KUKA KRL program: MyProgram_326().src

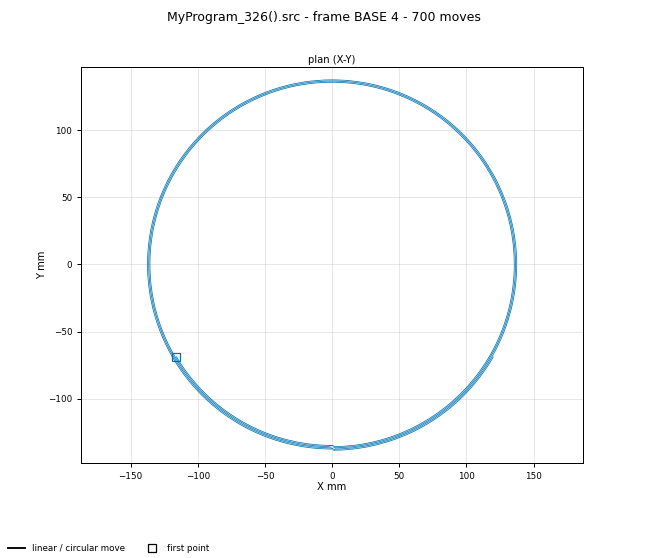
[picture p0: tool path of MyProgram_326().src in frame BASE 4, 700 of 700 moves have a stored position in this frame; points joined in program order, loops and branches not executed]
&ACCESS RVP
&REL 1
&PARAM TEMPLATE = C:\KRC\Roboter\Template\vorgabe
&PARAM EDITMASK = *
DEF MyProgram_326()
; ---- Setting reference (Base) ----
$BASE = BASE_DATA[4]

; --------------------------
; ---- Setting tool (TCP) ----
$TOOL = TOOL_DATA[3]
; --------------------------

$VEL.CP = VEL_APROX_PRINT
Startdeposition()
$VEL.CP = VEL_PRINT
LIN {X -115.9349,Y -68.7238,Z 187,A -143.6936,B 2.3952,C 0.2174,E1 2.2694,E2 236.7794} C_DIS
LIN {X -113.7532,Y -72.2781,Z 187,A -141.7842,B 2.3949,C 0.2211,E1 2.2723,E2 234.8528} C_DIS
LIN {X -111.2945,Y -76.0091,Z 187,A -139.8146,B 2.3945,C 0.2252,E1 2.2754,E2 232.8747} C_DIS
LIN {X -108.8442,Y -79.4786,Z 187,A -137.9392,B 2.3942,C 0.229,E1 2.2785,E2 230.9906} C_DIS
LIN {X -106.312,Y -82.8349,Z 187,A -136.0382,B 2.3938,C 0.2325,E1 2.2817,E2 229.0753} C_DIS
LIN {X -103.5544,Y -86.2576,Z 187,A -134.0833,B 2.3935,C 0.2361,E1 2.2852,E2 227.1095} C_DIS
LIN {X -101.6499,Y -88.4933,Z 187,A -132.7971,B 2.3932,C 0.2385,E1 2.2876,E2 225.8186} C_DIS
LIN {X -98.2627,Y -92.2405,Z 187,A -130.5399,B 2.3928,C 0.2423,E1 2.2919,E2 223.5473} C_DIS
LIN {X -95.1682,Y -95.4297,Z 187,A -128.6658,B 2.3925,C 0.2459,E1 2.2955,E2 221.6755} C_DIS
LIN {X -92.3122,Y -98.195,Z 187,A -126.8323,B 2.3922,C 0.2485,E1 2.2993,E2 219.8233} C_DIS
LIN {X -88.9634,Y -101.2395,Z 187,A -124.8002,B 2.3919,C 0.2515,E1 2.3036,E2 217.7772} C_DIS
LIN {X -85.547,Y -104.1421,Z 187,A -122.818,B 2.3916,C 0.2544,E1 2.3078,E2 215.785} C_DIS
LIN {X -81.9072,Y -107.0279,Z 187,A -120.8161,B 2.3913,C 0.2574,E1 2.3123,E2 213.7795} C_DIS
LIN {X -78.1832,Y -109.778,Z 187,A -118.865,B 2.3909,C 0.2605,E1 2.3167,E2 211.8306} C_DIS
LIN {X -75.0371,Y -111.952,Z 187,A -117.1257,B 2.3907,C 0.2623,E1 2.3207,E2 210.0763} C_DIS
LIN {X -71.5976,Y -114.1827,Z 187,A -115.4752,B 2.3904,C 0.2651,E1 2.3246,E2 208.438} C_DIS
LIN {X -68.7293,Y -115.9316,Z 187,A -113.528,B 2.3904,C 0.2648,E1 2.3294,E2 206.422} C_DIS
LIN {X -65.4366,Y -117.8212,Z 187,A -112.1847,B 2.3901,C 0.2678,E1 2.3326,E2 205.1144} C_DIS
LIN {X -61.68,Y -119.8297,Z 187,A -110.3476,B 2.3899,C 0.2698,E1 2.3372,E2 203.2735} C_DIS
LIN {X -58.7156,Y -121.3102,Z 187,A -108.8853,B 2.3898,C 0.271,E1 2.3409,E2 201.804} C_DIS
LIN {X -55.1373,Y -122.9761,Z 187,A -107.3291,B 2.3895,C 0.2732,E1 2.3448,E2 200.2636} C_DIS
LIN {X -52.5704,Y -124.0969,Z 187,A -105.9692,B 2.3895,C 0.2736,E1 2.3484,E2 198.881} C_DIS
LIN {X -49.184,Y -125.4763,Z 187,A -104.5101,B 2.3893,C 0.2753,E1 2.3521,E2 197.4343} C_DIS
LIN {X -45.9049,Y -126.7124,Z 187,A -103.0422,B 2.3891,C 0.2766,E1 2.356,E2 195.9689} C_DIS
LIN {X -42.7913,Y -127.7975,Z 187,A -101.597,B 2.3891,C 0.2774,E1 2.3598,E2 194.5176} C_DIS
LIN {X -40.0237,Y -128.6924,Z 187,A -100.359,B 2.3889,C 0.2782,E1 2.3631,E2 193.2791} C_DIS
LIN {X -36.5749,Y -129.7136,Z 187,A -98.7075,B 2.3889,C 0.2785,E1 2.3676,E2 191.611} C_DIS
LIN {X -32.9446,Y -130.6827,Z 187,A -97.0537,B 2.3889,C 0.2791,E1 2.3721,E2 189.9491} C_DIS
LIN {X -28.7479,Y -131.6698,Z 187,A -95.2714,B 2.3887,C 0.2801,E1 2.3769,E2 188.173} C_DIS
LIN {X -25.8135,Y -132.2771,Z 187,A -94.096,B 2.3887,C 0.2811,E1 2.3801,E2 187.0102} C_DIS
LIN {X -22.474,Y -132.8846,Z 187,A -92.5645,B 2.3887,C 0.2811,E1 2.3844,E2 185.4665} C_DIS
LIN {X -19.2693,Y -133.3868,Z 187,A -91.2519,B 2.3885,C 0.2817,E1 2.388,E2 184.1621} C_DIS
LIN {X -16.6253,Y -133.7436,Z 187,A -89.7338,B 2.3888,C 0.2798,E1 2.3923,E2 182.5925} C_DIS
LIN {X -11.5747,Y -134.2737,Z 187,A -87.959,B 2.3885,C 0.282,E1 2.3972,E2 180.868} C_DIS
LIN {X -8.5498,Y -134.5003,Z 187,A -86.5532,B 2.3885,C 0.2813,E1 2.4011,E2 179.4461} C_DIS
LIN {X -4.5816,Y -134.6953,Z 187,A -84.6494,B 2.3887,C 0.28,E1 2.4065,E2 177.513} C_DIS
LIN {X 0.9674,Y -134.7656,Z 187,A -83.2917,B 2.3881,C 0.2853,E1 2.41,E2 176.2871} C_DIS
Enddeposition()
LIN {X 0.9674,Y -134.7656,Z 187,A -83.292,B 2.3881,C 0.2853,E1 2.41,E2 176.2874} C_DIS
Startdeposition()
$VEL.CP = VEL_PRINT
LIN {X -3.9628,Y -135.6135,Z 187,A -85.1649,B 2.3882,C 0.2857,E1 2.4049,E2 178.1637} C_DIS
LIN {X -8.7995,Y -135.3863,Z 187,A -87.2259,B 2.3882,C 0.2859,E1 2.3991,E2 180.2278} C_DIS
LIN {X -12.7611,Y -135.0698,Z 187,A -89.7573,B 2.3876,C 0.2904,E1 2.3917,E2 182.8726} C_DIS
LIN {X -18.8714,Y -134.3525,Z 187,A -91.335,B 2.3883,C 0.2846,E1 2.3877,E2 184.3165} C_DIS
LIN {X -22.2434,Y -133.8352,Z 187,A -92.9879,B 2.3883,C 0.2854,E1 2.3831,E2 185.9982} C_DIS
LIN {X -25.7756,Y -133.2003,Z 187,A -94.5307,B 2.3883,C 0.285,E1 2.3788,E2 187.5451} C_DIS
LIN {X -29.9469,Y -132.3248,Z 187,A -96.3766,B 2.3883,C 0.2846,E1 2.3737,E2 189.3977} C_DIS
LIN {X -33.3901,Y -131.4978,Z 187,A -97.8597,B 2.3884,C 0.2838,E1 2.3697,E2 190.8796} C_DIS
LIN {X -36.7075,Y -130.6107,Z 187,A -99.3356,B 2.3885,C 0.2831,E1 2.3657,E2 192.3593} C_DIS
LIN {X -39.8775,Y -129.678,Z 187,A -100.6939,B 2.3886,C 0.2821,E1 2.3621,E2 193.7131} C_DIS
LIN {X -43.502,Y -128.5091,Z 187,A -102.3444,B 2.3887,C 0.2812,E1 2.3577,E2 195.3697} C_DIS
LIN {X -46.7066,Y -127.3797,Z 187,A -103.9429,B 2.3887,C 0.2808,E1 2.3534,E2 196.9901} C_DIS
LIN {X -50.9164,Y -125.7541,Z 187,A -105.7795,B 2.389,C 0.2789,E1 2.3487,E2 198.8179} C_DIS
LIN {X -54.0938,Y -124.4205,Z 187,A -107.2232,B 2.3892,C 0.2775,E1 2.345,E2 200.2604} C_DIS
LIN {X -57.1308,Y -123.0554,Z 187,A -108.6725,B 2.3893,C 0.2763,E1 2.3413,E2 201.7157} C_DIS
LIN {X -60.2592,Y -121.5542,Z 187,A -110.2095,B 2.3895,C 0.2751,E1 2.3374,E2 203.2623} C_DIS
LIN {X -64.2646,Y -119.487,Z 187,A -112.1562,B 2.3897,C 0.2731,E1 2.3325,E2 205.215} C_DIS
LIN {X -68.1062,Y -117.3398,Z 187,A -114.0242,B 2.3899,C 0.2709,E1 2.328,E2 207.0844} C_DIS
LIN {X -70.5754,Y -115.8722,Z 187,A -115.3814,B 2.39,C 0.2699,E1 2.3247,E2 208.4608} C_DIS
LIN {X -74.248,Y -113.5539,Z 187,A -117.2873,B 2.3903,C 0.2677,E1 2.3202,E2 210.3762} C_DIS
LIN {X -77.9286,Y -111.06,Z 187,A -119.2336,B 2.3906,C 0.2652,E1 2.3157,E2 212.3315} C_DIS
LIN {X -81.702,Y -108.3137,Z 187,A -121.2278,B 2.3909,C 0.2623,E1 2.3112,E2 214.3288} C_DIS
LIN {X -85.3873,Y -105.4331,Z 187,A -123.2774,B 2.3912,C 0.2594,E1 2.3067,E2 216.3881} C_DIS
LIN {X -88.8431,Y -102.5384,Z 187,A -125.2696,B 2.3915,C 0.2565,E1 2.3024,E2 218.3917} C_DIS
LIN {X -92.1943,Y -99.536,Z 187,A -127.2609,B 2.3918,C 0.2535,E1 2.2983,E2 220.3947} C_DIS
LIN {X -95.6007,Y -96.2682,Z 187,A -129.2474,B 2.3922,C 0.2498,E1 2.2943,E2 222.3802} C_DIS
LIN {X -98.4455,Y -93.3578,Z 187,A -131.4518,B 2.3924,C 0.2481,E1 2.2899,E2 224.6474} C_DIS
LIN {X -101.1671,Y -90.4008,Z 187,A -132.8605,B 2.3929,C 0.2438,E1 2.2874,E2 226.0185} C_DIS
LIN {X -104.2937,Y -86.7756,Z 187,A -134.9741,B 2.3932,C 0.2399,E1 2.2835,E2 228.1437} C_DIS
LIN {X -106.9935,Y -83.4242,Z 187,A -136.9228,B 2.3936,C 0.2365,E1 2.2801,E2 230.109} C_DIS
LIN {X -109.7743,Y -79.7289,Z 187,A -138.8973,B 2.394,C 0.2323,E1 2.2768,E2 232.0858} C_DIS
LIN {X -112.1941,Y -76.2865,Z 187,A -140.7335,B 2.3944,C 0.2285,E1 2.2739,E2 233.9292} C_DIS
LIN {X -114.4798,Y -72.8121,Z 187,A -142.6332,B 2.3947,C 0.2249,E1 2.271,E2 235.8469} C_DIS
LIN {X -116.6638,Y -69.2581,Z 187,A -144.7082,B 2.395,C 0.2217,E1 2.2679,E2 237.9617} C_DIS
LIN {X -118.2978,Y -66.4282,Z 187,A -145.964,B 2.3953,C 0.218,E1 2.2662,E2 239.2012} C_DIS
LIN {X -120.6007,Y -62.1484,Z 187,A -147.9412,B 2.3958,C 0.2129,E1 2.2636,E2 241.168} C_DIS
LIN {X -122.5743,Y -58.1567,Z 187,A -150.0373,B 2.3962,C 0.2088,E1 2.261,E2 243.2909} C_DIS
LIN {X -123.964,Y -55.132,Z 187,A -151.5191,B 2.3964,C 0.2054,E1 2.2593,E2 244.782} C_DIS
LIN {X -125.2998,Y -52.0247,Z 187,A -153.0319,B 2.3967,C 0.202,E1 2.2577,E2 246.305} C_DIS
LIN {X -126.6482,Y -48.6526,Z 187,A -154.7922,B 2.397,C 0.1986,E1 2.2559,E2 248.0935} C_DIS
LIN {X -127.9399,Y -45.1497,Z 187,A -156.5936,B 2.3973,C 0.195,E1 2.2542,E2 249.9229} C_DIS
LIN {X -128.9765,Y -42.0967,Z 187,A -158.0447,B 2.3976,C 0.1916,E1 2.2529,E2 251.3847} C_DIS
LIN {X -129.9685,Y -38.9282,Z 187,A -159.2035,B 2.3979,C 0.1873,E1 2.252,E2 252.512} C_DIS
LIN {X -130.8694,Y -35.7812,Z 187,A -160.6496,B 2.3982,C 0.1838,E1 2.2509,E2 253.9656} C_DIS
LIN {X -131.648,Y -32.7985,Z 187,A -162.038,B 2.3985,C 0.1804,E1 2.2499,E2 255.3642} C_DIS
LIN {X -132.4349,Y -29.4649,Z 187,A -163.7721,B 2.3987,C 0.1771,E1 2.2488,E2 257.134} C_DIS
LIN {X -133.2686,Y -25.4182,Z 187,A -165.4874,B 2.3991,C 0.1723,E1 2.2479,E2 258.8446} C_DIS
LIN {X -133.8544,Y -22.1283,Z 187,A -166.9599,B 2.3993,C 0.1685,E1 2.2472,E2 260.3241} C_DIS
LIN {X -134.4724,Y -17.9986,Z 187,A -168.8934,B 2.3996,C 0.164,E1 2.2464,E2 262.278} C_DIS
LIN {X -134.9012,Y -14.4335,Z 187,A -170.4596,B 2.3999,C 0.1599,E1 2.2459,E2 263.8496} C_DIS
LIN {X -135.2524,Y -10.6773,Z 187,A -172.3062,B 2.4002,C 0.156,E1 2.2455,E2 265.7271} C_DIS
LIN {X -135.4975,Y -6.8626,Z 187,A -173.8406,B 2.4005,C 0.1513,E1 2.2452,E2 267.2504} C_DIS
LIN {X -135.6224,Y -3.6402,Z 187,A -175.3722,B 2.4007,C 0.1478,E1 2.2451,E2 268.8024} C_DIS
LIN {X -135.6686,Y 0.848,Z 187,A -177.4173,B 2.401,C 0.1428,E1 2.2451,E2 270.8649} C_DIS
LIN {X -135.5766,Y 5.0694,Z 187,A -179.2202,B 2.4013,C 0.1378,E1 2.2452,E2 272.6692} C_DIS
LIN {X -135.3986,Y 8.5997,Z 187,A 179.0923,B 2.4015,C 0.1341,E1 2.2455,E2 274.3799} C_DIS
LIN {X -135.0608,Y 12.8544,Z 187,A 177.2514,B 2.4018,C 0.1291,E1 2.2459,E2 276.2243} C_DIS
LIN {X -134.6352,Y 16.7471,Z 187,A 175.3469,B 2.402,C 0.125,E1 2.2466,E2 278.1587} C_DIS
LIN {X -134.0771,Y 20.7351,Z 187,A 173.6992,B 2.4022,C 0.1202,E1 2.2472,E2 279.7987} C_DIS
LIN {X -133.5071,Y 24.1356,Z 187,A 172.1443,B 2.4024,C 0.1163,E1 2.248,E2 281.3648} C_DIS
LIN {X -132.7502,Y 28.0068,Z 187,A 169.9053,B 2.4026,C 0.113,E1 2.2493,E2 283.6729} C_DIS
LIN {X -131.8555,Y 31.9492,Z 187,A 168.5558,B 2.4028,C 0.1075,E1 2.2501,E2 284.9775} C_DIS
LIN {X -130.7952,Y 36.048,Z 187,A 165.9871,B 2.403,C 0.1044,E1 2.2521,E2 287.6399} C_DIS
LIN {X -129.3359,Y 40.9742,Z 187,A 164.5936,B 2.4033,C 0.0969,E1 2.2531,E2 288.9376} C_DIS
LIN {X -127.5776,Y 46.1576,Z 187,A 161.9652,B 2.4035,C 0.0915,E1 2.2556,E2 291.603} C_DIS
LIN {X -126.3033,Y 49.5398,Z 187,A 160.3094,B 2.4036,C 0.0878,E1 2.2572,E2 293.2736} C_DIS
LIN {X -124.9481,Y 52.8669,Z 187,A 158.075,B 2.4037,C 0.0855,E1 2.2598,E2 295.5934} C_DIS
LIN {X -122.9929,Y 57.2661,Z 187,A 156.5825,B 2.4039,C 0.0791,E1 2.2614,E2 297.0193} C_DIS
LIN {X -121.4822,Y 60.4052,Z 187,A 154.9035,B 2.404,C 0.0759,E1 2.2635,E2 298.7224} C_DIS
LIN {X -119.3862,Y 64.4522,Z 187,A 152.861,B 2.4042,C 0.0715,E1 2.2662,E2 300.7777} C_DIS
LIN {X -117.1973,Y 68.3524,Z 187,A 150.879,B 2.4042,C 0.0672,E1 2.2689,E2 302.7696} C_DIS
LIN {X -114.9211,Y 72.1134,Z 187,A 148.8626,B 2.4044,C 0.0632,E1 2.2719,E2 304.8037} C_DIS
LIN {X -111.6182,Y 77.1273,Z 187,A 146.0159,B 2.4045,C 0.0582,E1 2.2764,E2 307.6857} C_DIS
LIN {X -109.6336,Y 79.9229,Z 187,A 144.7535,B 2.4046,C 0.0545,E1 2.2785,E2 308.925} C_DIS
LIN {X -106.9745,Y 83.4473,Z 187,A 142.2883,B 2.4046,C 0.052,E1 2.2828,E2 311.46} C_DIS
LIN {X -104.0006,Y 87.126,Z 187,A 140.202,B 2.4047,C 0.0481,E1 2.2866,E2 313.5554} C_DIS
LIN {X -100.9239,Y 90.6724,Z 187,A 138.6902,B 2.4048,C 0.0428,E1 2.2893,E2 315.01} C_DIS
LIN {X -98.31,Y 93.5003,Z 187,A 136.8199,B 2.4048,C 0.0403,E1 2.2929,E2 316.9082} C_DIS
LIN {X -95.6937,Y 96.1759,Z 187,A 135.4271,B 2.405,C 0.0367,E1 2.2956,E2 318.2775} C_DIS
LIN {X -92.8995,Y 98.8778,Z 187,A 133.5688,B 2.405,C 0.0343,E1 2.2994,E2 320.1604} C_DIS
LIN {X -89.6074,Y 101.8709,Z 187,A 131.576,B 2.405,C 0.0313,E1 2.3036,E2 322.1653} C_DIS
LIN {X -86.1634,Y 104.8002,Z 187,A 129.7207,B 2.405,C 0.0279,E1 2.3075,E2 324.0129} C_DIS
LIN {X -80.2847,Y 109.3683,Z 187,A 126.7291,B 2.4051,C 0.0224,E1 2.3141,E2 326.9844} C_DIS
LIN {X -76.1837,Y 112.2637,Z 187,A 123.8354,B 2.4051,C 0.0217,E1 2.321,E2 329.9676} C_DIS
LIN {X -72.8163,Y 114.4771,Z 187,A 122.4348,B 2.4051,C 0.0183,E1 2.3242,E2 331.3318} C_DIS
LIN {X -69.1162,Y 116.7484,Z 187,A 120.5233,B 2.4051,C 0.0162,E1 2.3288,E2 333.2513} C_DIS
LIN {X -65.2576,Y 118.948,Z 187,A 117.9931,B 2.4051,C 0.0162,E1 2.3352,E2 335.8566} C_DIS
LIN {X -60.518,Y 121.4265,Z 187,A 116.5144,B 2.4052,C 0.0108,E1 2.3386,E2 337.2428} C_DIS
LIN {X -58.2312,Y 122.5387,Z 187,A 115.279,B 2.4052,C 0.0102,E1 2.3418,E2 338.4965} C_DIS
LIN {X -54.4677,Y 124.2588,Z 187,A 113.4333,B 2.4052,C 0.0088,E1 2.3465,E2 340.3527} C_DIS
LIN {X -50.9024,Y 125.7598,Z 187,A 111.1789,B 2.4052,C 0.0098,E1 2.3526,E2 342.6782} C_DIS
LIN {X -46.0846,Y 127.6039,Z 187,A 109.9279,B 2.4052,C 0.0043,E1 2.3555,E2 343.8198} C_DIS
LIN {X -42.3967,Y 128.8771,Z 187,A 107.7771,B 2.4052,C 0.0051,E1 2.3614,E2 346.0287} C_DIS
LIN {X -37.6699,Y 130.3371,Z 187,A 105.8675,B 2.4052,C 0.003,E1 2.3664,E2 347.916} C_DIS
LIN {X -34.8474,Y 131.1192,Z 187,A 104.5925,B 2.4052,C 0.0024,E1 2.3699,E2 349.1948} C_DIS
LIN {X -31.2485,Y 132.0244,Z 187,A 102.8608,B 2.4052,C 0.0024,E1 2.3747,E2 350.9449} C_DIS
LIN {X -26.9842,Y 132.9604,Z 187,A 101.1901,B 2.4052,C 0.0008,E1 2.3792,E2 352.5944} C_DIS
LIN {X -23.511,Y 133.6189,Z 187,A 99.6757,B 2.4052,C 0.0004,E1 2.3833,E2 354.1105} C_DIS
LIN {X -20.3204,Y 134.1413,Z 187,A 98.2387,B 2.4052,C 0.0004,E1 2.3873,E2 355.5553} C_DIS
LIN {X -16.0807,Y 134.7147,Z 187,A 96.1013,B 2.4052,C 0.0016,E1 2.3934,E2 357.7302} C_DIS
LIN {X -12.5247,Y 135.0924,Z 187,A 94.9072,B 2.4052,C -0.0001,E1 2.3966,E2 358.8869} C_DIS
LIN {X -8.6066,Y 135.3981,Z 187,A 93.2159,B 2.4052,C -0.0001,E1 2.4013,E2 360.5811} C_DIS
LIN {X -4.3157,Y 135.6037,Z 187,A 91.0044,B 2.4052,C 0.0021,E1 2.4076,E2 362.8381} C_DIS
LIN {X -0.2001,Y 135.6722,Z 187,A 89.4814,B 2.4052,C 0.0013,E1 2.4118,E2 364.3353} C_DIS
LIN {X 4.4585,Y 135.5997,Z 187,A 87.63,B 2.4052,C 0.0011,E1 2.417,E2 366.1724} C_DIS
LIN {X 8.4613,Y 135.4071,Z 187,A 86.0874,B 2.4052,C 0.0009,E1 2.4212,E2 367.6968} C_DIS
LIN {X 15.1854,Y 134.8202,Z 187,A 83.301,B 2.4052,C 0.0018,E1 2.429,E2 370.4748} C_DIS
LIN {X 17.74,Y 134.5063,Z 187,A 82.1957,B 2.4052,C 0.0024,E1 2.432,E2 371.5819} C_DIS
LIN {X 20.9884,Y 134.0379,Z 187,A 80.8084,B 2.4052,C 0.0032,E1 2.4359,E2 372.9689} C_DIS
LIN {X 24.959,Y 133.3564,Z 187,A 79.041,B 2.4052,C 0.0047,E1 2.4408,E2 374.7436} C_DIS
LIN {X 28.736,Y 132.5928,Z 187,A 77.5792,B 2.4052,C 0.005,E1 2.4447,E2 376.1854} C_DIS
LIN {X 31.8243,Y 131.8856,Z 187,A 76.2094,B 2.4052,C 0.0062,E1 2.4485,E2 377.5586} C_DIS
LIN {X 35.2871,Y 131.002,Z 187,A 74.7633,B 2.4052,C 0.0072,E1 2.4524,E2 378.9968} C_DIS
LIN {X 38.2039,Y 130.1808,Z 187,A 73.4505,B 2.4052,C 0.0086,E1 2.4559,E2 380.3132} C_DIS
LIN {X 42.0771,Y 128.9836,Z 187,A 71.816,B 2.4052,C 0.0098,E1 2.4602,E2 381.9383} C_DIS
LIN {X 44.9784,Y 127.9993,Z 187,A 70.5582,B 2.4052,C 0.011,E1 2.4635,E2 383.1916} C_DIS
LIN {X 47.9664,Y 126.9091,Z 187,A 69.2726,B 2.4052,C 0.0121,E1 2.4669,E2 384.4701} C_DIS
LIN {X 50.8513,Y 125.7804,Z 187,A 67.9156,B 2.4052,C 0.014,E1 2.4704,E2 385.8326} C_DIS
LIN {X 53.8514,Y 124.5253,Z 187,A 66.6364,B 2.4052,C 0.0151,E1 2.4737,E2 387.1005} C_DIS
LIN {X 56.9703,Y 123.1296,Z 187,A 65.1674,B 2.4052,C 0.0171,E1 2.4774,E2 388.5724} C_DIS
LIN {X 60.5139,Y 121.4285,Z 187,A 63.6187,B 2.4052,C 0.0186,E1 2.4813,E2 390.1077} C_DIS
LIN {X 63.3422,Y 119.9765,Z 187,A 62.3011,B 2.4052,C 0.0204,E1 2.4846,E2 391.4223} C_DIS
LIN {X 67.314,Y 117.796,Z 187,A 60.3527,B 2.4052,C 0.0235,E1 2.4893,E2 393.3747} C_DIS
LIN {X 71.0157,Y 115.6021,Z 187,A 58.5807,B 2.4051,C 0.026,E1 2.4936,E2 395.1412} C_DIS
LIN {X 74.6336,Y 113.3,Z 187,A 56.8868,B 2.4051,C 0.0282,E1 2.4975,E2 396.8212} C_DIS
LIN {X 78.0611,Y 110.9665,Z 187,A 55.1364,B 2.4051,C 0.0312,E1 2.5015,E2 398.5714} C_DIS
LIN {X 81.6721,Y 108.3362,Z 187,A 53.3465,B 2.405,C 0.0339,E1 2.5055,E2 400.3499} C_DIS
LIN {X 85.0579,Y 105.6988,Z 187,A 51.5712,B 2.405,C 0.0369,E1 2.5094,E2 402.1208} C_DIS
LIN {X 88.6943,Y 102.6666,Z 187,A 49.6611,B 2.4049,C 0.0401,E1 2.5135,E2 404.0204} C_DIS
LIN {X 94.9612,Y 96.8991,Z 187,A 46.4531,B 2.4049,C 0.0445,E1 2.52,E2 407.1821} C_DIS
LIN {X 98.902,Y 92.8738,Z 187,A 44.2564,B 2.4047,C 0.0481,E1 2.5242,E2 409.3573} C_DIS
LIN {X 101.9491,Y 89.5188,Z 187,A 42.0713,B 2.4047,C 0.0543,E1 2.5283,E2 411.5755} C_DIS
LIN {X 104.8825,Y 86.0628,Z 187,A 40.2699,B 2.4045,C 0.0577,E1 2.5315,E2 413.3636} C_DIS
LIN {X 107.6305,Y 82.6003,Z 187,A 38.4736,B 2.4045,C 0.0614,E1 2.5346,E2 415.1518} C_DIS
LIN {X 110.4322,Y 78.815,Z 187,A 36.6067,B 2.4044,C 0.0651,E1 2.5377,E2 417.0044} C_DIS
LIN {X 112.993,Y 75.0982,Z 187,A 34.791,B 2.4042,C 0.0689,E1 2.5405,E2 418.8096} C_DIS
LIN {X 115.0942,Y 71.8362,Z 187,A 33.2238,B 2.4042,C 0.0723,E1 2.5428,E2 420.3686} C_DIS
LIN {X 118.0799,Y 66.8158,Z 187,A 31.1357,B 2.404,C 0.0754,E1 2.5457,E2 422.4112} C_DIS
LIN {X 120.2703,Y 62.7828,Z 187,A 29.0959,B 2.4039,C 0.0811,E1 2.5484,E2 424.464} C_DIS
LIN {X 122.1618,Y 59.02,Z 187,A 27.2234,B 2.4037,C 0.0864,E1 2.5507,E2 426.3487} C_DIS
LIN {X 124.1968,Y 54.6112,Z 187,A 25.3425,B 2.4035,C 0.0903,E1 2.5529,E2 428.2097} C_DIS
LIN {X 126.2546,Y 49.6649,Z 187,A 23.1073,B 2.4033,C 0.096,E1 2.5552,E2 430.4424} C_DIS
LIN {X 128.1998,Y 44.4,Z 187,A 21.07,B 2.4032,C 0.0996,E1 2.5571,E2 432.4397} C_DIS
LIN {X 129.4223,Y 40.7039,Z 187,A 19.4383,B 2.403,C 0.104,E1 2.5585,E2 434.0707} C_DIS
LIN {X 130.6041,Y 36.7312,Z 187,A 17.8545,B 2.4028,C 0.1073,E1 2.5597,E2 435.6347} C_DIS
LIN {X 131.5365,Y 33.2376,Z 187,A 16.4565,B 2.4027,C 0.1105,E1 2.5607,E2 437.0174} C_DIS
LIN {X 132.432,Y 29.4775,Z 187,A 14.7904,B 2.4025,C 0.1152,E1 2.5617,E2 438.6886} C_DIS
LIN {X 133.2757,Y 25.3814,Z 187,A 13.2258,B 2.4023,C 0.1184,E1 2.5626,E2 440.2289} C_DIS
LIN {X 133.9255,Y 21.7018,Z 187,A 11.7123,B 2.4021,C 0.1223,E1 2.5633,E2 441.7354} C_DIS
LIN {X 134.4857,Y 17.8971,Z 187,A 9.8427,B 2.4018,C 0.1288,E1 2.564,E2 443.6363} C_DIS
LIN {X 134.9422,Y 14.0524,Z 187,A 8.6825,B 2.4018,C 0.1295,E1 2.5643,E2 444.7383} C_DIS
LIN {X 135.491,Y 6.9913,Z 187,A 6.0861,B 2.4015,C 0.1346,E1 2.5649,E2 447.287} C_DIS
LIN {X 135.6682,Y -0.9083,Z 187,A 2.5964,B 2.4008,C 0.1452,E1 2.565,E2 450.798} C_DIS
LIN {X 135.5747,Y -5.1196,Z 187,A 1.0097,B 2.4006,C 0.1486,E1 2.5649,E2 452.3615} C_DIS
LIN {X 135.397,Y -8.6255,Z 187,A -0.3873,B 2.4004,C 0.152,E1 2.5647,E2 453.7487} C_DIS
LIN {X 134.661,Y -16.5307,Z 187,A -3.4884,B 2.4,C 0.1593,E1 2.5639,E2 456.8202} C_DIS
LIN {X 134.2616,Y -19.5075,Z 187,A -4.7227,B 2.3997,C 0.1626,E1 2.5634,E2 458.051} C_DIS
LIN {X 133.7683,Y -22.6444,Z 187,A -5.977,B 2.3995,C 0.1656,E1 2.5628,E2 459.2952} C_DIS
LIN {X 133.2154,Y -25.6965,Z 187,A -7.2797,B 2.3993,C 0.1691,E1 2.5621,E2 460.5979} C_DIS
LIN {X 132.4021,Y -29.6084,Z 187,A -8.9226,B 2.399,C 0.1734,E1 2.5612,E2 462.2364} C_DIS
LIN {X 131.4838,Y -33.4454,Z 187,A -10.426,B 2.3987,C 0.1766,E1 2.5602,E2 463.7202} C_DIS
LIN {X 130.5312,Y -36.9918,Z 187,A -11.8717,B 2.3985,C 0.18,E1 2.5591,E2 465.1535} C_DIS
LIN {X 129.3987,Y -40.7778,Z 187,A -13.6763,B 2.3981,C 0.1856,E1 2.5576,E2 466.9768} C_DIS
LIN {X 127.308,Y -46.9017,Z 187,A -16.1603,B 2.3977,C 0.1909,E1 2.5553,E2 469.4309} C_DIS
LIN {X 125.8906,Y -50.5779,Z 187,A -17.7333,B 2.3974,C 0.1945,E1 2.5537,E2 470.9934} C_DIS
LIN {X 124.4088,Y -54.1208,Z 187,A -19.1471,B 2.3972,C 0.197,E1 2.5522,E2 472.3817} C_DIS
LIN {X 123.0265,Y -57.1935,Z 187,A -20.5226,B 2.3969,C 0.2003,E1 2.5506,E2 473.7521} C_DIS
LIN {X 121.5101,Y -60.3486,Z 187,A -21.9477,B 2.3966,C 0.2037,E1 2.5489,E2 475.1715} C_DIS
LIN {X 119.4628,Y -64.3096,Z 187,A -24.3097,B 2.3958,C 0.2124,E1 2.5457,E2 477.5966} C_DIS
LIN {X 116.9512,Y -68.7713,Z 187,A -25.5312,B 2.396,C 0.2101,E1 2.5442,E2 478.6985} C_DIS
LIN {X 114.3355,Y -73.0375,Z 187,A -28.6356,B 2.3949,C 0.2232,E1 2.5394,E2 481.9324} C_DIS
LIN {X 110.6412,Y -78.5223,Z 187,A -30.4697,B 2.3949,C 0.2222,E1 2.5366,E2 483.6451} C_DIS
LIN {X 108.0948,Y -81.992,Z 187,A -32.2772,B 2.3946,C 0.2263,E1 2.5336,E2 485.4527} C_DIS
LIN {X 105.2053,Y -85.6678,Z 187,A -34.1452,B 2.3942,C 0.2299,E1 2.5304,E2 487.3084} C_DIS
LIN {X 102.3834,Y -89.0211,Z 187,A -36.0805,B 2.3938,C 0.2347,E1 2.5268,E2 489.2562} C_DIS
LIN {X 100.2438,Y -91.4241,Z 187,A -37.1305,B 2.3938,C 0.2352,E1 2.5249,E2 490.2669} C_DIS
LIN {X 97.4141,Y -94.4328,Z 187,A -39.2703,B 2.393,C 0.242,E1 2.5207,E2 492.4597} C_DIS
LIN {X 94.2721,Y -97.5698,Z 187,A -40.4564,B 2.3932,C 0.2405,E1 2.5185,E2 493.5572} C_DIS
LIN {X 90.4673,Y -101.1075,Z 187,A -42.7155,B 2.3927,C 0.2455,E1 2.5138,E2 495.8266} C_DIS
LIN {X 87.3717,Y -103.7945,Z 187,A -44.776,B 2.3921,C 0.2513,E1 2.5093,E2 497.9316} C_DIS
LIN {X 84.1771,Y -106.4023,Z 187,A -46.1439,B 2.3921,C 0.2517,E1 2.5064,E2 499.2519} C_DIS
LIN {X 79.101,Y -110.2278,Z 187,A -48.3876,B 2.3919,C 0.2533,E1 2.5015,E2 501.4396} C_DIS
LIN {X 76.6141,Y -111.9704,Z 187,A -49.9277,B 2.3914,C 0.2574,E1 2.4979,E2 503.0147} C_DIS
LIN {X 73.1785,Y -114.2453,Z 187,A -51.7754,B 2.391,C 0.2611,E1 2.4935,E2 504.8779} C_DIS
LIN {X 67.2661,Y -117.8231,Z 187,A -54.4025,B 2.3907,C 0.2636,E1 2.4873,E2 507.4687} C_DIS
LIN {X 63.9396,Y -119.6616,Z 187,A -56.0519,B 2.3904,C 0.2663,E1 2.4832,E2 509.1252} C_DIS
LIN {X 59.4866,Y -121.9353,Z 187,A -57.9157,B 2.3904,C 0.2676,E1 2.4787,E2 510.9576} C_DIS
LIN {X 56.5818,Y -123.3093,Z 187,A -59.2528,B 2.3901,C 0.2693,E1 2.4753,E2 512.2931} C_DIS
LIN {X 53.6805,Y -124.5992,Z 187,A -60.5925,B 2.3899,C 0.271,E1 2.4718,E2 513.6335} C_DIS
LIN {X 50.2075,Y -126.0399,Z 187,A -62.1103,B 2.3898,C 0.2724,E1 2.4679,E2 515.1431} C_DIS
LIN {X 46.9999,Y -127.2712,Z 187,A -63.8691,B 2.3893,C 0.2762,E1 2.4632,E2 516.9437} C_DIS
LIN {X 43.6451,Y -128.4614,Z 187,A -65.0058,B 2.3894,C 0.2754,E1 2.4603,E2 518.0329} C_DIS
LIN {X 39.49,Y -129.7966,Z 187,A -66.7731,B 2.3893,C 0.2768,E1 2.4556,E2 519.7912} C_DIS
LIN {X 36.4093,Y -130.6941,Z 187,A -68.1122,B 2.3891,C 0.278,E1 2.452,E2 521.1291} C_DIS
LIN {X 33.1081,Y -131.5694,Z 187,A -69.5462,B 2.389,C 0.2792,E1 2.4482,E2 522.5629} C_DIS
LIN {X 29.8653,Y -132.3434,Z 187,A -71.0114,B 2.3888,C 0.2807,E1 2.4441,E2 524.0366} C_DIS
LIN {X 25.7649,Y -133.2023,Z 187,A -72.9884,B 2.3885,C 0.2834,E1 2.4386,E2 526.0421} C_DIS
LIN {X 22.501,Y -133.7922,Z 187,A -74.116,B 2.3885,C 0.2826,E1 2.4356,E2 527.1344} C_DIS
LIN {X 18.9431,Y -134.3423,Z 187,A -75.5797,B 2.3885,C 0.2832,E1 2.4316,E2 528.5914} C_DIS
LIN {X 15.2144,Y -134.8171,Z 187,A -77.6825,B 2.388,C 0.2871,E1 2.4256,E2 530.7634} C_DIS
LIN {X 10.6687,Y -135.2516,Z 187,A -79.1807,B 2.3882,C 0.2854,E1 2.4215,E2 532.2057} C_DIS
LIN {X 4.3047,Y -135.604,Z 187,A -81.607,B 2.3883,C 0.2847,E1 2.4148,E2 534.5981} C_DIS
LIN {X 0.9595,Y -135.6572,Z 187,A -83.6177,B 2.3879,C 0.2885,E1 2.409,E2 536.6884} C_DIS
Enddeposition()
LIN {X 0.9595,Y -135.6572,Z 187,A -83.6179,B 2.3879,C 0.2885,E1 2.409,E2 536.6887} C_DIS
Startdeposition()
$VEL.CP = VEL_PRINT
LIN {X 1.7111,Y -136.5613,Z 187,A -81.4555,B 2.402,C 0.2794,E1 2.4287,E2 534.3043} C_DIS
LIN {X 7.3621,Y -136.3732,Z 187,A -79.8542,B 2.4015,C 0.2833,E1 2.4328,E2 532.8067} C_DIS
LIN {X 15.3195,Y -135.7107,Z 187,A -76.5489,B 2.4017,C 0.2821,E1 2.442,E2 529.5059} C_DIS
LIN {X 21.4398,Y -134.8784,Z 187,A -73.6016,B 2.4021,C 0.2782,E1 2.4503,E2 526.5089} C_DIS
LIN {X 25.0218,Y -134.2604,Z 187,A -72.525,B 2.4019,C 0.2801,E1 2.4531,E2 525.4922} C_DIS
LIN {X 28.8804,Y -133.482,Z 187,A -70.8156,B 2.4021,C 0.2784,E1 2.4578,E2 523.7739} C_DIS
LIN {X 32.2398,Y -132.7109,Z 187,A -69.4087,B 2.4022,C 0.2775,E1 2.4616,E2 522.3714} C_DIS
LIN {X 35.3465,Y -131.9172,Z 187,A -68.0779,B 2.4023,C 0.2764,E1 2.4652,E2 521.0417} C_DIS
LIN {X 38.3774,Y -131.0674,Z 187,A -66.7391,B 2.4025,C 0.275,E1 2.4688,E2 519.6996} C_DIS
LIN {X 41.9265,Y -129.9762,Z 187,A -65.256,B 2.4026,C 0.2739,E1 2.4728,E2 518.2256} C_DIS
LIN {X 45.7216,Y -128.6912,Z 187,A -63.316,B 2.403,C 0.2702,E1 2.478,E2 516.2495} C_DIS
LIN {X 48.8823,Y -127.5241,Z 187,A -62.3104,B 2.4029,C 0.2714,E1 2.4805,E2 515.298} C_DIS
LIN {X 51.4277,Y -126.5181,Z 187,A -61.1083,B 2.4031,C 0.2696,E1 2.4836,E2 514.0879} C_DIS
LIN {X 55.1509,Y -124.9411,Z 187,A -59.3502,B 2.4034,C 0.267,E1 2.4882,E2 512.3203} C_DIS
LIN {X 59.063,Y -123.1384,Z 187,A -57.6965,B 2.4035,C 0.2657,E1 2.4923,E2 510.686} C_DIS
LIN {X 62.4196,Y -121.4722,Z 187,A -56.1737,B 2.4037,C 0.2638,E1 2.4961,E2 509.1687} C_DIS
LIN {X 65.7667,Y -119.6951,Z 187,A -54.1995,B 2.4043,C 0.2586,E1 2.5011,E2 507.1416} C_DIS
LIN {X 69.3539,Y -117.6524,Z 187,A -52.8403,B 2.4043,C 0.2586,E1 2.5042,E2 505.8314} C_DIS
LIN {X 73.0609,Y -115.3869,Z 187,A -51.3357,B 2.4043,C 0.2581,E1 2.5077,E2 504.3682} C_DIS
LIN {X 75.7242,Y -113.6568,Z 187,A -49.8412,B 2.4047,C 0.2546,E1 2.5112,E2 502.851} C_DIS
LIN {X 79.2365,Y -111.2368,Z 187,A -47.6235,B 2.4054,C 0.2482,E1 2.5164,E2 500.5742} C_DIS
LIN {X 83.1442,Y -108.3471,Z 187,A -46.3925,B 2.4051,C 0.2507,E1 2.519,E2 499.4504} C_DIS
LIN {X 87.1314,Y -105.1671,Z 187,A -44.0955,B 2.4057,C 0.2455,E1 2.524,E2 497.1307} C_DIS
LIN {X 90.4809,Y -102.2996,Z 187,A -42.0428,B 2.4062,C 0.2403,E1 2.5284,E2 495.0494} C_DIS
LIN {X 93.1725,Y -99.8544,Z 187,A -40.8796,B 2.4062,C 0.24,E1 2.5307,E2 493.9336} C_DIS
LIN {X 97.558,Y -95.5743,Z 187,A -38.4711,B 2.4066,C 0.236,E1 2.5354,E2 491.5448} C_DIS
LIN {X 100.2598,Y -92.737,Z 187,A -36.652,B 2.4071,C 0.2311,E1 2.5389,E2 489.701} C_DIS
LIN {X 103.9359,Y -88.5967,Z 187,A -34.5555,B 2.4074,C 0.2278,E1 2.5427,E2 487.6328} C_DIS
LIN {X 106.3687,Y -85.6605,Z 187,A -33.0631,B 2.4077,C 0.225,E1 2.5453,E2 486.1535} C_DIS
LIN {X 109.1682,Y -82.0632,Z 187,A -31.2312,B 2.408,C 0.2213,E1 2.5484,E2 484.3307} C_DIS
LIN {X 111.7059,Y -78.5737,Z 187,A -28.5647,B 2.409,C 0.2099,E1 2.5529,E2 481.5484} C_DIS
LIN {X 115.858,Y -72.3115,Z 187,A -26.6054,B 2.4088,C 0.2122,E1 2.5556,E2 479.7459} C_DIS
LIN {X 120.5925,Y -64.1043,Z 187,A -22.8584,B 2.4095,C 0.2042,E1 2.5608,E2 476.0261} C_DIS
LIN {X 122.0473,Y -61.2901,Z 187,A -21.5503,B 2.4098,C 0.201,E1 2.5624,E2 474.7198} C_DIS
LIN {X 123.3079,Y -58.7081,Z 187,A -20.3629,B 2.41,C 0.198,E1 2.5638,E2 473.5338} C_DIS
LIN {X 124.9421,Y -55.1488,Z 187,A -18.6429,B 2.4104,C 0.1931,E1 2.5658,E2 471.8025} C_DIS
LIN {X 126.8348,Y -50.6419,Z 187,A -16.9035,B 2.4107,C 0.1903,E1 2.5676,E2 470.1024} C_DIS
LIN {X 128.1505,Y -47.2173,Z 187,A -15.4391,B 2.4109,C 0.1869,E1 2.569,E2 468.6467} C_DIS
LIN {X 129.9784,Y -41.9196,Z 187,A -13.1435,B 2.4114,C 0.181,E1 2.5711,E2 466.3566} C_DIS
LIN {X 131.1154,Y -38.2136,Z 187,A -11.6624,B 2.4116,C 0.1779,E1 2.5723,E2 464.8933} C_DIS
LIN {X 132.0379,Y -34.8941,Z 187,A -10.281,B 2.4119,C 0.1745,E1 2.5733,E2 463.5192} C_DIS
LIN {X 132.9666,Y -31.1772,Z 187,A -8.6927,B 2.4122,C 0.1702,E1 2.5743,E2 461.9323} C_DIS
LIN {X 133.8258,Y -27.243,Z 187,A -7.1822,B 2.4124,C 0.1671,E1 2.5752,E2 460.4437} C_DIS
LIN {X 134.4451,Y -24.0011,Z 187,A -5.8768,B 2.4126,C 0.1639,E1 2.5758,E2 459.1477} C_DIS
LIN {X 135.0452,Y -20.3627,Z 187,A -4.4462,B 2.4128,C 0.1606,E1 2.5764,E2 457.7311} C_DIS
LIN {X 135.5461,Y -16.7063,Z 187,A -2.4424,B 2.4134,C 0.1524,E1 2.5771,E2 455.6672} C_DIS
LIN {X 136.0358,Y -12.0909,Z 187,A -0.9663,B 2.4134,C 0.151,E1 2.5775,E2 454.2509} C_DIS
LIN {X 136.3216,Y -8.2478,Z 187,A 0.9687,B 2.4139,C 0.1437,E1 2.5779,E2 452.2737} C_DIS
LIN {X 136.531,Y -3.3314,Z 187,A 2.3067,B 2.4139,C 0.1441,E1 2.5779,E2 451.0282} C_DIS
LIN {X 136.493,Y 4.6586,Z 187,A 5.5447,B 2.4144,C 0.1357,E1 2.5779,E2 447.8031} C_DIS
LIN {X 136.0117,Y 12.3635,Z 187,A 8.5357,B 2.4147,C 0.1287,E1 2.5773,E2 444.842} C_DIS
LIN {X 135.3189,Y 18.463,Z 187,A 11.0034,B 2.4151,C 0.1224,E1 2.5765,E2 442.3867} C_DIS
LIN {X 134.767,Y 22.1255,Z 187,A 12.5765,B 2.4153,C 0.1179,E1 2.5758,E2 440.8103} C_DIS
LIN {X 134.037,Y 26.1902,Z 187,A 14.097,B 2.4154,C 0.1149,E1 2.575,E2 439.3158} C_DIS
LIN {X 133.4356,Y 29.0952,Z 187,A 15.3049,B 2.4156,C 0.1118,E1 2.5743,E2 438.1119} C_DIS
LIN {X 132.7245,Y 32.1833,Z 187,A 16.5451,B 2.4157,C 0.1089,E1 2.5735,E2 436.8824} C_DIS
LIN {X 131.8379,Y 35.6441,Z 187,A 17.9555,B 2.4159,C 0.1056,E1 2.5725,E2 435.4824} C_DIS
LIN {X 130.9376,Y 38.8208,Z 187,A 19.26,B 2.4159,C 0.1025,E1 2.5715,E2 434.1874} C_DIS
LIN {X 130.0387,Y 41.7307,Z 187,A 20.4969,B 2.4161,C 0.0994,E1 2.5705,E2 432.955} C_DIS
LIN {X 128.9159,Y 45.0812,Z 187,A 21.9329,B 2.4163,C 0.0958,E1 2.5692,E2 431.5242} C_DIS
LIN {X 126.347,Y 51.8463,Z 187,A 24.6986,B 2.4165,C 0.09,E1 2.5665,E2 428.7913} C_DIS
LIN {X 125.1579,Y 54.6554,Z 187,A 26.1013,B 2.4166,C 0.0857,E1 2.5649,E2 427.3728} C_DIS
LIN {X 123.4406,Y 58.4304,Z 187,A 27.5222,B 2.4167,C 0.0838,E1 2.5633,E2 425.9911} C_DIS
LIN {X 122.367,Y 60.6451,Z 187,A 28.6539,B 2.4168,C 0.0804,E1 2.5618,E2 424.8467} C_DIS
LIN {X 120.3986,Y 64.4688,Z 187,A 30.4467,B 2.417,C 0.0759,E1 2.5595,E2 423.0547} C_DIS
LIN {X 117.8102,Y 69.0852,Z 187,A 32.6837,B 2.4171,C 0.0703,E1 2.5564,E2 420.815} C_DIS
LIN {X 115.1231,Y 73.4758,Z 187,A 34.6098,B 2.4172,C 0.0669,E1 2.5536,E2 418.9175} C_DIS
LIN {X 112.9493,Y 76.7758,Z 187,A 36.1731,B 2.4173,C 0.0637,E1 2.5512,E2 417.3654} C_DIS
LIN {X 110.4811,Y 80.2868,Z 187,A 37.8892,B 2.4174,C 0.0601,E1 2.5484,E2 415.6593} C_DIS
LIN {X 108.0057,Y 83.587,Z 187,A 39.5589,B 2.4175,C 0.0567,E1 2.5456,E2 413.9968} C_DIS
LIN {X 105.0871,Y 87.228,Z 187,A 41.4108,B 2.4175,C 0.0531,E1 2.5423,E2 412.1576} C_DIS
LIN {X 102.1073,Y 90.6985,Z 187,A 43.2618,B 2.4177,C 0.0494,E1 2.5389,E2 410.3146} C_DIS
LIN {X 97.8824,Y 95.2426,Z 187,A 45.6812,B 2.4177,C 0.0453,E1 2.5343,E2 407.9175} C_DIS
LIN {X 94.8798,Y 98.2336,Z 187,A 48.017,B 2.4179,C 0.0375,E1 2.5295,E2 405.5127} C_DIS
LIN {X 90.9143,Y 101.915,Z 187,A 49.5679,B 2.4179,C 0.0384,E1 2.5265,E2 404.0502} C_DIS
LIN {X 87.6602,Y 104.7268,Z 187,A 51.3533,B 2.4179,C 0.035,E1 2.5227,E2 402.267} C_DIS
LIN {X 84.1438,Y 107.5728,Z 187,A 53.1914,B 2.4179,C 0.032,E1 2.5187,E2 400.4362} C_DIS
LIN {X 80.5099,Y 110.3193,Z 187,A 55.0677,B 2.4179,C 0.0288,E1 2.5145,E2 398.5641} C_DIS
LIN {X 76.8398,Y 112.906,Z 187,A 56.8667,B 2.418,C 0.0262,E1 2.5104,E2 396.7754} C_DIS
LIN {X 73.0303,Y 115.4063,Z 187,A 58.6353,B 2.418,C 0.0241,E1 2.5062,E2 395.0242} C_DIS
LIN {X 69.5368,Y 117.5449,Z 187,A 60.391,B 2.418,C 0.0211,E1 2.502,E2 393.2642} C_DIS
LIN {X 65.1313,Y 120.0417,Z 187,A 62.3769,B 2.418,C 0.0189,E1 2.4972,E2 391.2952} C_DIS
LIN {X 62.1801,Y 121.5942,Z 187,A 63.7527,B 2.4181,C 0.0171,E1 2.4938,E2 389.9223} C_DIS
LIN {X 58.8043,Y 123.262,Z 187,A 65.262,B 2.4181,C 0.0154,E1 2.49,E2 388.4216} C_DIS
LIN {X 55.3051,Y 124.8722,Z 187,A 66.7767,B 2.4181,C 0.014,E1 2.4862,E2 386.9195} C_DIS
LIN {X 52.0494,Y 126.2645,Z 187,A 68.2326,B 2.4181,C 0.0123,E1 2.4824,E2 385.4674} C_DIS
LIN {X 49.1364,Y 127.4254,Z 187,A 69.5335,B 2.4181,C 0.0109,E1 2.4791,E2 384.1684} C_DIS
LIN {X 46.0937,Y 128.557,Z 187,A 70.8544,B 2.4181,C 0.0096,E1 2.4756,E2 382.8527} C_DIS
LIN {X 42.9867,Y 129.6289,Z 187,A 72.2015,B 2.4181,C 0.0084,E1 2.472,E2 381.5097} C_DIS
LIN {X 39.8283,Y 130.6339,Z 187,A 73.5665,B 2.4181,C 0.0072,E1 2.4684,E2 380.1481} C_DIS
LIN {X 36.3246,Y 131.652,Z 187,A 75.2016,B 2.4181,C 0.0051,E1 2.464,E2 378.5008} C_DIS
LIN {X 32.1963,Y 132.7214,Z 187,A 76.8756,B 2.4181,C 0.0043,E1 2.4595,E2 376.8411} C_DIS
LIN {X 28.4582,Y 133.5732,Z 187,A 78.3633,B 2.4181,C 0.0038,E1 2.4554,E2 375.3684} C_DIS
LIN {X 25.5528,Y 134.1589,Z 187,A 79.5809,B 2.4181,C 0.0031,E1 2.4521,E2 374.1541} C_DIS
LIN {X 22.5708,Y 134.6927,Z 187,A 80.8896,B 2.4181,C 0.0021,E1 2.4485,E2 372.8413} C_DIS
LIN {X 19.3172,Y 135.1976,Z 187,A 82.2726,B 2.4181,C 0.0013,E1 2.4447,E2 371.4585} C_DIS
LIN {X 15.5639,Y 135.6824,Z 187,A 84.0656,B 2.4181,C -0.0007,E1 2.4396,E2 369.6416} C_DIS
LIN {X 9.5704,Y 136.2356,Z 187,A 86.4599,B 2.4181,C -0.001,E1 2.433,E2 367.2638} C_DIS
LIN {X 2.3895,Y 136.5501,Z 187,A 89.1711,B 2.4181,C -0.0001,E1 2.4255,E2 364.5903} C_DIS
LIN {X -4.4737,Y 136.4993,Z 187,A 92.3383,B 2.4181,C -0.002,E1 2.4166,E2 361.3901} C_DIS
LIN {X -10.656,Y 136.1563,Z 187,A 95.4894,B 2.4181,C -0.0047,E1 2.4076,E2 358.1736} C_DIS
LIN {X -15.912,Y 135.6409,Z 187,A 96.804,B 2.4181,C 0,E1 2.4042,E2 356.9682} C_DIS
LIN {X -19.0508,Y 135.2357,Z 187,A 98.4161,B 2.4181,C -0.0011,E1 2.3997,E2 355.3229} C_DIS
LIN {X -22.6162,Y 134.6851,Z 187,A 99.8604,B 2.4181,C -0.0003,E1 2.3957,E2 353.8876} C_DIS
LIN {X -25.8244,Y 134.1069,Z 187,A 101.2868,B 2.4181,C -0.0001,E1 2.3917,E2 352.4548} C_DIS
LIN {X -29.1045,Y 133.4337,Z 187,A 102.6611,B 2.4181,C 0.0006,E1 2.388,E2 351.085} C_DIS
LIN {X -32.2545,Y 132.7073,Z 187,A 104.015,B 2.4181,C 0.0013,E1 2.3843,E2 349.732} C_DIS
LIN {X -35.3235,Y 131.9234,Z 187,A 105.4384,B 2.4181,C 0.0016,E1 2.3804,E2 348.2981} C_DIS
LIN {X -40.0845,Y 130.5555,Z 187,A 107.2804,B 2.4181,C 0.004,E1 2.3756,E2 346.4855} C_DIS
LIN {X -43.2693,Y 129.5348,Z 187,A 108.9402,B 2.4181,C 0.0039,E1 2.3711,E2 344.7959} C_DIS
LIN {X -46.6043,Y 128.3729,Z 187,A 110.438,B 2.4181,C 0.005,E1 2.3671,E2 343.2971} C_DIS
LIN {X -53.3887,Y 125.7052,Z 187,A 113.541,B 2.4181,C 0.0076,E1 2.3591,E2 340.1908} C_DIS
LIN {X -56.1684,Y 124.486,Z 187,A 114.8738,B 2.4181,C 0.0086,E1 2.3556,E2 338.8516} C_DIS
LIN {X -59.8369,Y 122.7657,Z 187,A 117.3569,B 2.4181,C 0.0074,E1 2.3492,E2 336.2751} C_DIS
LIN {X -64.9341,Y 120.1483,Z 187,A 119.204,B 2.4181,C 0.0124,E1 2.3448,E2 334.497} C_DIS
LIN {X -69.0194,Y 117.8489,Z 187,A 121.4822,B 2.4181,C 0.0138,E1 2.3392,E2 332.1825} C_DIS
LIN {X -72.2797,Y 115.8778,Z 187,A 122.8512,B 2.4181,C 0.0168,E1 2.336,E2 330.8422} C_DIS
LIN {X -75.5749,Y 113.7565,Z 187,A 124.4689,B 2.4181,C 0.0192,E1 2.3322,E2 329.2288} C_DIS
LIN {X -78.7877,Y 111.555,Z 187,A 126.2007,B 2.4181,C 0.0213,E1 2.3282,E2 327.4863} C_DIS
LIN {X -82.1708,Y 109.087,Z 187,A 128.7045,B 2.4181,C 0.0216,E1 2.3224,E2 324.893} C_DIS
LIN {X -86.6961,Y 105.5268,Z 187,A 130.339,B 2.4181,C 0.0282,E1 2.3191,E2 323.3552} C_DIS
LIN {X -89.2771,Y 103.3521,Z 187,A 131.9587,B 2.418,C 0.03,E1 2.3156,E2 321.7118} C_DIS
LIN {X -92.4831,Y 100.4932,Z 187,A 133.8652,B 2.418,C 0.0329,E1 2.3116,E2 319.794} C_DIS
LIN {X -95.6311,Y 97.5023,Z 187,A 135.8326,B 2.4179,C 0.0358,E1 2.3076,E2 317.8102} C_DIS
LIN {X -98.1531,Y 94.963,Z 187,A 137.2895,B 2.4179,C 0.0389,E1 2.3048,E2 316.3598} C_DIS
LIN {X -100.9599,Y 91.9737,Z 187,A 139.0537,B 2.4178,C 0.0421,E1 2.3014,E2 314.5915} C_DIS
LIN {X -104.377,Y 88.0772,Z 187,A 142.1144,B 2.4178,C 0.0441,E1 2.2957,E2 311.4238} C_DIS
LIN {X -108.0418,Y 83.5403,Z 187,A 143.8518,B 2.4176,C 0.0514,E1 2.2928,E2 309.7754} C_DIS
LIN {X -110.3858,Y 80.4182,Z 187,A 146.1123,B 2.4176,C 0.0533,E1 2.289,E2 307.4398} C_DIS
LIN {X -112.9098,Y 76.8337,Z 187,A 147.9692,B 2.4175,C 0.0574,E1 2.2861,E2 305.582} C_DIS
LIN {X -115.1229,Y 73.4762,Z 187,A 149.1405,B 2.4174,C 0.0627,E1 2.2844,E2 304.4753} C_DIS
LIN {X -116.7931,Y 70.7911,Z 187,A 150.805,B 2.4173,C 0.0649,E1 2.2819,E2 302.7704} C_DIS
LIN {X -118.9798,Y 67.051,Z 187,A 152.699,B 2.4172,C 0.0691,E1 2.2792,E2 300.8683} C_DIS
LIN {X -121.0947,Y 63.1481,Z 187,A 154.5628,B 2.417,C 0.0736,E1 2.2768,E2 299.0056} C_DIS
LIN {X -122.5792,Y 60.2149,Z 187,A 156.1,B 2.417,C 0.0767,E1 2.2749,E2 297.4499} C_DIS
LIN {X -124.9505,Y 55.1298,Z 187,A 158.9641,B 2.4168,C 0.0814,E1 2.2715,E2 294.5243} C_DIS
LIN {X -126.4914,Y 51.4939,Z 187,A 160.1065,B 2.4166,C 0.0869,E1 2.2704,E2 293.4469} C_DIS
LIN {X -128.0663,Y 47.4421,Z 187,A 162.4742,B 2.4165,C 0.0904,E1 2.2679,E2 291.013} C_DIS
LIN {X -129.6336,Y 42.9728,Z 187,A 164.3277,B 2.4163,C 0.096,E1 2.2663,E2 289.1776} C_DIS
LIN {X -131.3829,Y 37.2869,Z 187,A 166.8104,B 2.416,C 0.1027,E1 2.2643,E2 286.6984} C_DIS
LIN {X -132.0609,Y 34.8079,Z 187,A 168.1705,B 2.4159,C 0.105,E1 2.2633,E2 285.3038} C_DIS
LIN {X -133.0094,Y 30.9899,Z 187,A 170.3482,B 2.4157,C 0.1083,E1 2.2619,E2 283.0611} C_DIS
LIN {X -133.9031,Y 26.8633,Z 187,A 171.7332,B 2.4155,C 0.114,E1 2.2611,E2 281.7259} C_DIS
LIN {X -134.5678,Y 23.3155,Z 187,A 173.4897,B 2.4153,C 0.1177,E1 2.2602,E2 279.94} C_DIS
LIN {X -135.2069,Y 19.2525,Z 187,A 175.1886,B 2.4151,C 0.1225,E1 2.2595,E2 278.2455} C_DIS
LIN {X -135.6252,Y 16.043,Z 187,A 176.5815,B 2.4149,C 0.1262,E1 2.259,E2 276.8492} C_DIS
LIN {X -135.9567,Y 12.9373,Z 187,A 178.0258,B 2.4147,C 0.1296,E1 2.2586,E2 275.3889} C_DIS
LIN {X -136.2953,Y 8.676,Z 187,A 179.9354,B 2.4144,C 0.1344,E1 2.2582,E2 273.4657} C_DIS
LIN {X -136.4789,Y 5.0203,Z 187,A -178.4658,B 2.4142,C 0.1386,E1 2.2581,E2 271.8599} C_DIS
LIN {X -136.5675,Y 0.9982,Z 187,A -176.6058,B 2.4139,C 0.1429,E1 2.258,E2 269.9791} C_DIS
LIN {X -136.5329,Y -3.2654,Z 187,A -174.6868,B 2.4137,C 0.1477,E1 2.258,E2 268.0447} C_DIS
LIN {X -136.3933,Y -6.9633,Z 187,A -173.1386,B 2.4134,C 0.152,E1 2.2583,E2 266.4979} C_DIS
LIN {X -136.171,Y -10.4551,Z 187,A -171.5861,B 2.4131,C 0.1559,E1 2.2586,E2 264.9354} C_DIS
LIN {X -135.9066,Y -13.4586,Z 187,A -170.2335,B 2.4129,C 0.1593,E1 2.2589,E2 263.5723} C_DIS
LIN {X -135.5009,Y -17.0737,Z 187,A -168.4676,B 2.4127,C 0.163,E1 2.2595,E2 261.7767} C_DIS
LIN {X -134.9763,Y -20.8078,Z 187,A -166.8838,B 2.4124,C 0.1674,E1 2.2602,E2 260.1934} C_DIS
LIN {X -134.3954,Y -24.279,Z 187,A -165.3584,B 2.4121,C 0.1713,E1 2.2609,E2 258.6625} C_DIS
LIN {X -133.7832,Y -27.4527,Z 187,A -163.9375,B 2.4118,C 0.1749,E1 2.2617,E2 257.234} C_DIS
LIN {X -133.1102,Y -30.5485,Z 187,A -162.4783,B 2.4116,C 0.1782,E1 2.2626,E2 255.7587} C_DIS
LIN {X -132.1792,Y -34.3626,Z 187,A -160.598,B 2.4113,C 0.1821,E1 2.2639,E2 253.8491} C_DIS
LIN {X -131.3895,Y -37.2633,Z 187,A -159.2844,B 2.4111,C 0.1854,E1 2.2649,E2 252.5294} C_DIS
LIN {X -129.0825,Y -44.6004,Z 187,A -155.9711,B 2.4104,C 0.1937,E1 2.2677,E2 249.2065} C_DIS
LIN {X -127.5278,Y -48.873,Z 187,A -154.0448,B 2.41,C 0.1986,E1 2.2696,E2 247.2785} C_DIS
LIN {X -126.5715,Y -51.2951,Z 187,A -152.8014,B 2.4098,C 0.201,E1 2.2709,E2 246.016} C_DIS
LIN {X -125.2057,Y -54.5448,Z 187,A -151.2113,B 2.4095,C 0.2045,E1 2.2727,E2 244.412} C_DIS
LIN {X -123.9012,Y -57.4453,Z 187,A -149.8183,B 2.4092,C 0.2077,E1 2.2743,E2 243.0117} C_DIS
LIN {X -122.3929,Y -60.5926,Z 187,A -148.2377,B 2.4089,C 0.211,E1 2.2763,E2 241.4165} C_DIS
LIN {X -120.2738,Y -64.7011,Z 187,A -146.1738,B 2.4086,C 0.2153,E1 2.279,E2 239.3369} C_DIS
LIN {X -117.6159,Y -69.4161,Z 187,A -143.9162,B 2.4081,C 0.2208,E1 2.2821,E2 237.0819} C_DIS
LIN {X -115.7108,Y -72.5478,Z 187,A -142.1384,B 2.4078,C 0.2237,E1 2.2848,E2 235.273} C_DIS
LIN {X -113.4084,Y -76.0962,Z 187,A -140.3153,B 2.4074,C 0.2275,E1 2.2876,E2 233.4439} C_DIS
LIN {X -110.8957,Y -79.7136,Z 187,A -138.3433,B 2.4071,C 0.2312,E1 2.2908,E2 231.456} C_DIS
LIN {X -108.4204,Y -83.0484,Z 187,A -136.5042,B 2.4068,C 0.2347,E1 2.2939,E2 229.6046} C_DIS
LIN {X -105.5532,Y -86.6638,Z 187,A -134.468,B 2.4064,C 0.2384,E1 2.2975,E2 227.5555} C_DIS
LIN {X -102.5906,Y -90.1517,Z 187,A -132.2996,B 2.4061,C 0.2415,E1 2.3015,E2 225.3543} C_DIS
LIN {X -98.7566,Y -94.3352,Z 187,A -130.1941,B 2.4055,C 0.2471,E1 2.3055,E2 223.2857} C_DIS
LIN {X -96.2089,Y -96.9322,Z 187,A -128.5709,B 2.4053,C 0.2496,E1 2.3087,E2 221.6499} C_DIS
LIN {X -94.4153,Y -98.6801,Z 187,A -127.3359,B 2.4051,C 0.2509,E1 2.3112,E2 220.3904} C_DIS
LIN {X -91.2177,Y -101.6433,Z 187,A -125.4247,B 2.4048,C 0.2538,E1 2.3152,E2 218.4684} C_DIS
LIN {X -87.8817,Y -104.541,Z 187,A -123.4856,B 2.4045,C 0.2566,E1 2.3194,E2 216.518} C_DIS
LIN {X -84.2698,Y -107.4738,Z 187,A -121.4933,B 2.4042,C 0.2596,E1 2.3237,E2 214.5205} C_DIS
LIN {X -80.6872,Y -110.189,Z 187,A -119.5347,B 2.4039,C 0.2622,E1 2.3281,E2 212.5521} C_DIS
LIN {X -77.0855,Y -112.7381,Z 187,A -117.6122,B 2.4036,C 0.2646,E1 2.3326,E2 210.6201} C_DIS
LIN {X -73.712,Y -114.972,Z 187,A -115.8438,B 2.4034,C 0.2667,E1 2.3367,E2 208.842} C_DIS
LIN {X -70.1107,Y -117.203,Z 187,A -113.9165,B 2.4032,C 0.2684,E1 2.3414,E2 206.8944} C_DIS
LIN {X -67.0404,Y -118.9858,Z 187,A -112.5111,B 2.403,C 0.2706,E1 2.3448,E2 205.5002} C_DIS
LIN {X -63.2413,Y -121.0457,Z 187,A -110.7421,B 2.4027,C 0.2728,E1 2.3491,E2 203.7369} C_DIS
LIN {X -60.177,Y -122.5979,Z 187,A -109.231,B 2.4026,C 0.2741,E1 2.353,E2 202.2162} C_DIS
LIN {X -56.9018,Y -124.1526,Z 187,A -107.7324,B 2.4024,C 0.2757,E1 2.3567,E2 200.7203} C_DIS
LIN {X -53.8884,Y -125.4895,Z 187,A -106.2988,B 2.4023,C 0.2768,E1 2.3604,E2 199.2797} C_DIS
LIN {X -50.6229,Y -126.8425,Z 187,A -104.8225,B 2.4021,C 0.2781,E1 2.3643,E2 197.8039} C_DIS
LIN {X -47.6687,Y -127.9814,Z 187,A -103.4599,B 2.4021,C 0.279,E1 2.3678,E2 196.4364} C_DIS
LIN {X -44.564,Y -129.0952,Z 187,A -102.0246,B 2.4019,C 0.2798,E1 2.3717,E2 194.9939} C_DIS
LIN {X -41.3249,Y -130.1684,Z 187,A -100.5936,B 2.4019,C 0.2808,E1 2.3755,E2 193.5625} C_DIS
LIN {X -38.203,Y -131.1185,Z 187,A -99.1962,B 2.4017,C 0.2815,E1 2.3792,E2 192.1609} C_DIS
LIN {X -35.0803,Y -131.9882,Z 187,A -97.8111,B 2.4017,C 0.2821,E1 2.383,E2 190.772} C_DIS
LIN {X -31.4894,Y -132.8917,Z 187,A -96.2919,B 2.4016,C 0.283,E1 2.3871,E2 189.257} C_DIS
LIN {X -28.5909,Y -133.5445,Z 187,A -95.0383,B 2.4016,C 0.2834,E1 2.3905,E2 188.002} C_DIS
LIN {X -25.4786,Y -134.173,Z 187,A -93.6352,B 2.4015,C 0.2835,E1 2.3944,E2 186.5889} C_DIS
LIN {X -21.584,Y -134.8561,Z 187,A -91.8284,B 2.4015,C 0.2831,E1 2.3994,E2 184.7614} C_DIS
LIN {X -13.1257,Y -135.9386,Z 187,A -88.6877,B 2.4012,C 0.2861,E1 2.408,E2 181.6784} C_DIS
LIN {X -6.2288,Y -136.4301,Z 187,A -85.5426,B 2.4014,C 0.2847,E1 2.4169,E2 178.4994} C_DIS
LIN {X -0.6916,Y -136.5692,Z 187,A -83.5209,B 2.4012,C 0.2861,E1 2.4225,E2 176.5175} C_DIS
LIN {X -0.6916,Y -136.5692,Z 187,A -83.5211,B 2.4012,C 0.2861,E1 2.4225,E2 176.5177} C_DIS
Enddeposition()
LIN {X 0.9725,Y -137.4642,Z 187,A -82.6771,B 2.405,C 0.2865,E1 2.4286,E2 175.6821} C_DIS
Startdeposition()
$VEL.CP = VEL_PRINT
LIN {X -2.0056,Y -137.4563,Z 187,A -84.1237,B 2.4048,C 0.2879,E1 2.4245,E2 177.1573} C_DIS
LIN {X -5.1499,Y -137.3742,Z 187,A -85.494,B 2.4048,C 0.2884,E1 2.4206,E2 178.5364} C_DIS
LIN {X -8.6019,Y -137.2012,Z 187,A -87.3634,B 2.4044,C 0.2909,E1 2.4152,E2 180.4643} C_DIS
LIN {X -11.8564,Y -136.9585,Z 187,A -88.4817,B 2.4046,C 0.2895,E1 2.4122,E2 181.5505} C_DIS
LIN {X -15.7733,Y -136.5635,Z 187,A -90.1626,B 2.4046,C 0.2895,E1 2.4075,E2 183.2376} C_DIS
LIN {X -19.9982,Y -136.0091,Z 187,A -92.2104,B 2.4045,C 0.2907,E1 2.4017,E2 185.3226} C_DIS
LIN {X -23.551,Y -135.4397,Z 187,A -93.4878,B 2.4047,C 0.2891,E1 2.3983,E2 186.5707} C_DIS
LIN {X -27.2369,Y -134.7452,Z 187,A -94.9342,B 2.4047,C 0.288,E1 2.3943,E2 188.0018} C_DIS
LIN {X -30.0907,Y -134.1376,Z 187,A -96.0582,B 2.4049,C 0.287,E1 2.3913,E2 189.1138} C_DIS
LIN {X -33.6649,Y -133.2845,Z 187,A -97.7406,B 2.4049,C 0.287,E1 2.3867,E2 190.8171} C_DIS
LIN {X -37.0299,Y -132.389,Z 187,A -99.1913,B 2.405,C 0.2863,E1 2.3827,E2 192.2681} C_DIS
LIN {X -40.234,Y -131.4506,Z 187,A -100.5772,B 2.4051,C 0.2854,E1 2.379,E2 193.6536} C_DIS
LIN {X -43.2527,Y -130.4886,Z 187,A -101.9395,B 2.4051,C 0.2847,E1 2.3754,E2 195.0219} C_DIS
LIN {X -46.144,Y -129.4952,Z 187,A -103.2677,B 2.4053,C 0.284,E1 2.3719,E2 196.3577} C_DIS
LIN {X -49.4866,Y -128.2545,Z 187,A -104.8217,B 2.4053,C 0.2832,E1 2.3678,E2 197.9211} C_DIS
LIN {X -52.6931,Y -126.9707,Z 187,A -106.1253,B 2.4056,C 0.2813,E1 2.3644,E2 199.2068} C_DIS
LIN {X -55.8597,Y -125.6097,Z 187,A -107.6791,B 2.4056,C 0.2805,E1 2.3604,E2 200.7766} C_DIS
LIN {X -58.9226,Y -124.2025,Z 187,A -109.2174,B 2.4058,C 0.2796,E1 2.3565,E2 202.333} C_DIS
LIN {X -62.1658,Y -122.611,Z 187,A -110.5618,B 2.4061,C 0.2773,E1 2.3532,E2 203.656} C_DIS
LIN {X -65.3566,Y -120.9429,Z 187,A -112.2902,B 2.4061,C 0.2766,E1 2.3488,E2 205.4152} C_DIS
LIN {X -68.694,Y -119.0787,Z 187,A -113.9503,B 2.4063,C 0.2749,E1 2.3448,E2 207.0844} C_DIS
LIN {X -72.4204,Y -116.8499,Z 187,A -115.813,B 2.4066,C 0.2728,E1 2.3403,E2 208.9544} C_DIS
LIN {X -76.2534,Y -114.3852,Z 187,A -117.7041,B 2.4069,C 0.2701,E1 2.3359,E2 210.8444} C_DIS
LIN {X -79.614,Y -112.0729,Z 187,A -119.4978,B 2.4071,C 0.268,E1 2.3317,E2 212.6506} C_DIS
LIN {X -83.0989,Y -109.5137,Z 187,A -121.3654,B 2.4074,C 0.2655,E1 2.3275,E2 214.527} C_DIS
LIN {X -86.6575,Y -106.7203,Z 187,A -123.3501,B 2.4077,C 0.2628,E1 2.3232,E2 216.5248} C_DIS
LIN {X -90.12,Y -103.8126,Z 187,A -125.2926,B 2.408,C 0.2598,E1 2.319,E2 218.4749} C_DIS
LIN {X -93.4697,Y -100.807,Z 187,A -127.2402,B 2.4083,C 0.2568,E1 2.315,E2 220.4319} C_DIS
LIN {X -96.2067,Y -98.1979,Z 187,A -129.1696,B 2.4085,C 0.2551,E1 2.311,E2 222.4079} C_DIS
LIN {X -98.9334,Y -95.4505,Z 187,A -130.2428,B 2.409,C 0.2502,E1 2.3091,E2 223.4094} C_DIS
LIN {X -103.4503,Y -90.5353,Z 187,A -133.4601,B 2.4094,C 0.2462,E1 2.3029,E2 226.6841} C_DIS
LIN {X -106.4732,Y -86.9598,Z 187,A -135.4761,B 2.4098,C 0.2423,E1 2.2993,E2 228.7081} C_DIS
LIN {X -109.1453,Y -83.5815,Z 187,A -137.3393,B 2.4102,C 0.2387,E1 2.2961,E2 230.5799} C_DIS
LIN {X -111.8166,Y -79.9726,Z 187,A -139.2984,B 2.4106,C 0.2349,E1 2.2928,E2 232.5501} C_DIS
LIN {X -114.3227,Y -76.3471,Z 187,A -141.2233,B 2.4109,C 0.231,E1 2.2898,E2 234.4861} C_DIS
LIN {X -116.727,Y -72.6179,Z 187,A -143.2001,B 2.4113,C 0.2272,E1 2.2868,E2 236.4791} C_DIS
LIN {X -119.0739,Y -68.7023,Z 187,A -145.1226,B 2.4117,C 0.2227,E1 2.2841,E2 238.4035} C_DIS
LIN {X -121.1326,Y -65.0035,Z 187,A -147.1211,B 2.412,C 0.2191,E1 2.2813,E2 240.432} C_DIS
LIN {X -123.1365,Y -61.1188,Z 187,A -148.8924,B 2.4125,C 0.2145,E1 2.2791,E2 242.1961} C_DIS
LIN {X -124.4882,Y -58.3195,Z 187,A -150.1777,B 2.4127,C 0.2113,E1 2.2776,E2 243.4796} C_DIS
LIN {X -126.0682,Y -54.817,Z 187,A -151.9617,B 2.4131,C 0.2077,E1 2.2755,E2 245.2866} C_DIS
LIN {X -127.4277,Y -51.5776,Z 187,A -153.4618,B 2.4134,C 0.2041,E1 2.2739,E2 246.7909} C_DIS
LIN {X -128.4031,Y -49.1042,Z 187,A -154.7972,B 2.4136,C 0.2018,E1 2.2726,E2 248.1553} C_DIS
LIN {X -129.8476,Y -45.1403,Z 187,A -156.258,B 2.414,C 0.1964,E1 2.2712,E2 249.5767} C_DIS
LIN {X -130.4199,Y -43.4589,Z 187,A -157.6417,B 2.414,C 0.1961,E1 2.2699,E2 251.0432} C_DIS
LIN {X -131.4666,Y -40.1819,Z 187,A -158.8399,B 2.4144,C 0.1917,E1 2.2689,E2 252.2104} C_DIS
LIN {X -132.6584,Y -36.059,Z 187,A -160.8183,B 2.4147,C 0.1874,E1 2.2674,E2 254.2124} C_DIS
LIN {X -133.5665,Y -32.5296,Z 187,A -162.3372,B 2.415,C 0.1833,E1 2.2664,E2 255.7305} C_DIS
LIN {X -134.3447,Y -29.1478,Z 187,A -163.8655,B 2.4153,C 0.1795,E1 2.2655,E2 257.2687} C_DIS
LIN {X -134.9907,Y -25.9927,Z 187,A -165.1682,B 2.4156,C 0.1757,E1 2.2648,E2 258.5655} C_DIS
LIN {X -135.4586,Y -23.4453,Z 187,A -166.6033,B 2.4157,C 0.1736,E1 2.264,E2 260.0458} C_DIS
LIN {X -136.1035,Y -19.3376,Z 187,A -168.2954,B 2.4161,C 0.1687,E1 2.2633,E2 261.7316} C_DIS
LIN {X -136.6249,Y -15.2325,Z 187,A -170.1505,B 2.4164,C 0.1642,E1 2.2627,E2 263.6023} C_DIS
LIN {X -136.9672,Y -11.7536,Z 187,A -171.5853,B 2.4167,C 0.1601,E1 2.2623,E2 265.0335} C_DIS
LIN {X -137.1722,Y -9.0736,Z 187,A -172.7563,B 2.4169,C 0.157,E1 2.2621,E2 266.2103} C_DIS
LIN {X -137.3507,Y -5.7519,Z 187,A -174.3666,B 2.4171,C 0.1537,E1 2.2619,E2 267.8482} C_DIS
LIN {X -137.4551,Y -2.0759,Z 187,A -175.9579,B 2.4174,C 0.1495,E1 2.2618,E2 269.446} C_DIS
LIN {X -137.4583,Y 1.8821,Z 187,A -177.6725,B 2.4176,C 0.145,E1 2.2618,E2 271.1679} C_DIS
LIN {X -137.3935,Y 4.6554,Z 187,A -179.0764,B 2.4178,C 0.1423,E1 2.2619,E2 272.6023} C_DIS
LIN {X -137.1919,Y 8.753,Z 187,A 179.1572,B 2.4181,C 0.1376,E1 2.2622,E2 274.3747} C_DIS
LIN {X -136.8632,Y 12.9085,Z 187,A 177.3696,B 2.4183,C 0.1329,E1 2.2626,E2 276.1674} C_DIS
LIN {X -136.4992,Y 16.3125,Z 187,A 175.9785,B 2.4185,C 0.1288,E1 2.2631,E2 277.5532} C_DIS
LIN {X -136.1717,Y 18.8609,Z 187,A 174.6375,B 2.4187,C 0.1264,E1 2.2636,E2 278.9274} C_DIS
LIN {X -135.5956,Y 22.6258,Z 187,A 173.0684,B 2.4189,C 0.122,E1 2.2643,E2 280.493} C_DIS
LIN {X -135.1118,Y 25.3592,Z 187,A 171.9678,B 2.4191,C 0.1186,E1 2.2648,E2 281.5859} C_DIS
LIN {X -134.6625,Y 27.6432,Z 187,A 170.7219,B 2.4191,C 0.1166,E1 2.2655,E2 282.8655} C_DIS
LIN {X -133.6645,Y 32.1229,Z 187,A 168.7577,B 2.4194,C 0.1115,E1 2.2668,E2 284.8348} C_DIS
LIN {X -132.6219,Y 36.1958,Z 187,A 166.7206,B 2.4196,C 0.1074,E1 2.2683,E2 286.9061} C_DIS
LIN {X -131.3993,Y 40.4018,Z 187,A 164.9206,B 2.4198,C 0.1024,E1 2.2697,E2 288.7016} C_DIS
LIN {X -130.0482,Y 44.5616,Z 187,A 163.1835,B 2.42,C 0.0974,E1 2.2712,E2 290.4268} C_DIS
LIN {X -128.8853,Y 47.8203,Z 187,A 161.4787,B 2.4201,C 0.0942,E1 2.2728,E2 292.163} C_DIS
LIN {X -127.6254,Y 51.087,Z 187,A 158.7321,B 2.4201,C 0.0934,E1 2.276,E2 295.0658} C_DIS
LIN {X -124.4165,Y 58.4745,Z 187,A 156.2453,B 2.4206,C 0.0829,E1 2.2787,E2 297.4445} C_DIS
LIN {X -122.6337,Y 62.1213,Z 187,A 154.8202,B 2.4207,C 0.078,E1 2.2804,E2 298.8356} C_DIS
LIN {X -120.9266,Y 65.387,Z 187,A 152.8845,B 2.4208,C 0.0752,E1 2.283,E2 300.8192} C_DIS
LIN {X -118.6887,Y 69.366,Z 187,A 150.8752,B 2.4209,C 0.0709,E1 2.2858,E2 302.8402} C_DIS
LIN {X -116.3803,Y 73.1727,Z 187,A 149.1402,B 2.4211,C 0.0662,E1 2.2883,E2 304.5591} C_DIS
LIN {X -114.6203,Y 75.9003,Z 187,A 147.4788,B 2.4211,C 0.0639,E1 2.2909,E2 306.2571} C_DIS
LIN {X -112.2218,Y 79.4032,Z 187,A 145.6785,B 2.4212,C 0.06,E1 2.2938,E2 308.0599} C_DIS
LIN {X -109.4696,Y 83.1574,Z 187,A 143.5878,B 2.4213,C 0.0562,E1 2.2973,E2 310.1674} C_DIS
LIN {X -106.5165,Y 86.9068,Z 187,A 141.4519,B 2.4214,C 0.0523,E1 2.3011,E2 312.3196} C_DIS
LIN {X -103.2725,Y 90.7387,Z 187,A 139.3741,B 2.4214,C 0.048,E1 2.3049,E2 314.3941} C_DIS
LIN {X -100.4249,Y 93.8801,Z 187,A 137.5503,B 2.4216,C 0.0446,E1 2.3083,E2 316.2235} C_DIS
LIN {X -97.2876,Y 97.1276,Z 187,A 135.5185,B 2.4216,C 0.0414,E1 2.3123,E2 318.2719} C_DIS
LIN {X -93.9493,Y 100.3604,Z 187,A 133.5439,B 2.4216,C 0.038,E1 2.3163,E2 320.2497} C_DIS
LIN {X -90.7008,Y 103.3058,Z 187,A 131.6133,B 2.4217,C 0.035,E1 2.3204,E2 322.1914} C_DIS
LIN {X -87.3187,Y 106.1799,Z 187,A 129.8675,B 2.4217,C 0.0316,E1 2.3241,E2 323.9233} C_DIS
LIN {X -84.0154,Y 108.8119,Z 187,A 127.9319,B 2.4217,C 0.0292,E1 2.3284,E2 325.8788} C_DIS
LIN {X -80.7032,Y 111.2904,Z 187,A 126.1365,B 2.4218,C 0.0268,E1 2.3325,E2 327.6815} C_DIS
LIN {X -76.9598,Y 113.9112,Z 187,A 124.1551,B 2.4218,C 0.0242,E1 2.337,E2 329.6708} C_DIS
LIN {X -73.3151,Y 116.2904,Z 187,A 122.3593,B 2.4218,C 0.0216,E1 2.3413,E2 331.4632} C_DIS
LIN {X -68.7402,Y 119.0519,Z 187,A 120.0527,B 2.4218,C 0.019,E1 2.3468,E2 333.7778} C_DIS
LIN {X -65.4035,Y 120.9177,Z 187,A 118.3645,B 2.4219,C 0.0174,E1 2.351,E2 335.4764} C_DIS
LIN {X -59.2469,Y 124.0476,Z 187,A 115.5348,B 2.4219,C 0.014,E1 2.3581,E2 338.2984} C_DIS
LIN {X -56.3449,Y 125.3926,Z 187,A 114.2854,B 2.4219,C 0.0123,E1 2.3612,E2 339.537} C_DIS
LIN {X -53.9036,Y 126.4631,Z 187,A 113.0473,B 2.4219,C 0.0117,E1 2.3644,E2 340.7895} C_DIS
LIN {X -50.4157,Y 127.8933,Z 187,A 111.4854,B 2.4219,C 0.0102,E1 2.3685,E2 342.3494} C_DIS
LIN {X -47.9613,Y 128.8325,Z 187,A 110.3646,B 2.4219,C 0.0094,E1 2.3714,E2 343.4726} C_DIS
LIN {X -44.7668,Y 129.9771,Z 187,A 108.8316,B 2.4219,C 0.0088,E1 2.3755,E2 345.0188} C_DIS
LIN {X -40.7394,Y 131.296,Z 187,A 107.1227,B 2.4219,C 0.0073,E1 2.38,E2 346.72} C_DIS
LIN {X -37.0064,Y 132.3956,Z 187,A 105.3901,B 2.4219,C 0.0068,E1 2.3847,E2 348.4648} C_DIS
LIN {X -33.2907,Y 133.3795,Z 187,A 103.7029,B 2.4219,C 0.0063,E1 2.3893,E2 350.1612} C_DIS
LIN {X -29.5555,Y 134.2567,Z 187,A 102.2941,B 2.4219,C 0.0047,E1 2.3931,E2 351.5466} C_DIS
LIN {X -25.9956,Y 134.9902,Z 187,A 100.667,B 2.4219,C 0.0047,E1 2.3976,E2 353.1862} C_DIS
LIN {X -23.0724,Y 135.5211,Z 187,A 99.3614,B 2.4219,C 0.0045,E1 2.4012,E2 354.4992} C_DIS
LIN {X -19.6048,Y 136.0654,Z 187,A 97.9632,B 2.4219,C 0.0038,E1 2.405,E2 355.889} C_DIS
LIN {X -15.7541,Y 136.5658,Z 187,A 96.0999,B 2.4219,C 0.0048,E1 2.4103,E2 357.7806} C_DIS
LIN {X -7.0475,Y 137.2898,Z 187,A 92.6946,B 2.4219,C 0.0034,E1 2.4197,E2 361.1562} C_DIS
LIN {X -3.7591,Y 137.4192,Z 187,A 91.2639,B 2.4219,C 0.0038,E1 2.4237,E2 362.5934} C_DIS
LIN {X 1.7263,Y 137.4609,Z 187,A 88.9076,B 2.4219,C 0.0046,E1 2.4304,E2 364.9571} C_DIS
LIN {X 9.1515,Y 137.1674,Z 187,A 85.862,B 2.4219,C 0.0052,E1 2.4388,E2 367.9954} C_DIS
LIN {X 12.4413,Y 136.9081,Z 187,A 84.4006,B 2.4219,C 0.0063,E1 2.4429,E2 369.4665} C_DIS
LIN {X 18.969,Y 136.1562,Z 187,A 81.8248,B 2.4219,C 0.0067,E1 2.45,E2 372.022} C_DIS
LIN {X 22.4713,Y 135.6214,Z 187,A 80.4223,B 2.4219,C 0.0072,E1 2.4539,E2 373.4152} C_DIS
LIN {X 25.6811,Y 135.0503,Z 187,A 79.1665,B 2.4219,C 0.0075,E1 2.4573,E2 374.6583} C_DIS
LIN {X 28.2789,Y 134.5323,Z 187,A 77.827,B 2.4219,C 0.0097,E1 2.4611,E2 376.0256} C_DIS
LIN {X 32.3608,Y 133.6072,Z 187,A 76.2598,B 2.4219,C 0.01,E1 2.4653,E2 377.5711} C_DIS
LIN {X 36.0145,Y 132.6702,Z 187,A 74.5881,B 2.4219,C 0.012,E1 2.4698,E2 379.2544} C_DIS
LIN {X 40.0734,Y 131.4998,Z 187,A 72.9986,B 2.4219,C 0.0126,E1 2.474,E2 380.823} C_DIS
LIN {X 42.9492,Y 130.5897,Z 187,A 71.7114,B 2.4219,C 0.0141,E1 2.4775,E2 382.1135} C_DIS
LIN {X 46.1449,Y 129.4949,Z 187,A 70.2717,B 2.4219,C 0.0158,E1 2.4813,E2 383.5568} C_DIS
LIN {X 49.5458,Y 128.2315,Z 187,A 69.0011,B 2.4219,C 0.016,E1 2.4845,E2 384.7981} C_DIS
LIN {X 52.7462,Y 126.9485,Z 187,A 67.4961,B 2.4219,C 0.0181,E1 2.4884,E2 386.3111} C_DIS
LIN {X 55.8933,Y 125.5946,Z 187,A 66.0264,B 2.4219,C 0.0202,E1 2.4922,E2 387.7855} C_DIS
LIN {X 60.09,Y 123.644,Z 187,A 64.1074,B 2.4219,C 0.0227,E1 2.4971,E2 389.7033} C_DIS
LIN {X 63.4456,Y 121.9546,Z 187,A 62.7024,B 2.4219,C 0.0239,E1 2.5005,E2 391.0887} C_DIS
LIN {X 66.2757,Y 120.4418,Z 187,A 61.2901,B 2.4219,C 0.0263,E1 2.504,E2 392.5099} C_DIS
LIN {X 70.1707,Y 118.2146,Z 187,A 59.5044,B 2.4219,C 0.0286,E1 2.5083,E2 394.2854} C_DIS
LIN {X 74.1024,Y 115.7903,Z 187,A 57.6469,B 2.4218,C 0.0313,E1 2.5127,E2 396.1347} C_DIS
LIN {X 77.8241,Y 113.3224,Z 187,A 55.9095,B 2.4218,C 0.0335,E1 2.5167,E2 397.8571} C_DIS
LIN {X 81.2104,Y 110.9211,Z 187,A 54.1743,B 2.4217,C 0.0366,E1 2.5206,E2 399.5929} C_DIS
LIN {X 84.6937,Y 108.2848,Z 187,A 52.4389,B 2.4217,C 0.0393,E1 2.5244,E2 401.318} C_DIS
LIN {X 88.1364,Y 105.5017,Z 187,A 50.6352,B 2.4216,C 0.0424,E1 2.5283,E2 403.1168} C_DIS
LIN {X 91.4547,Y 102.6388,Z 187,A 48.7787,B 2.4216,C 0.0462,E1 2.5322,E2 404.9771} C_DIS
LIN {X 95.0562,Y 99.3121,Z 187,A 46.9437,B 2.4215,C 0.0488,E1 2.5359,E2 406.7869} C_DIS
LIN {X 98.2781,Y 96.1249,Z 187,A 45.219,B 2.4215,C 0.0515,E1 2.5393,E2 408.4919} C_DIS
LIN {X 100.7301,Y 93.5523,Z 187,A 43.6718,B 2.4213,C 0.0551,E1 2.5422,E2 410.0473} C_DIS
LIN {X 103.9065,Y 90.0119,Z 187,A 41.8422,B 2.4213,C 0.0583,E1 2.5456,E2 411.8587} C_DIS
LIN {X 106.7076,Y 86.673,Z 187,A 40.0854,B 2.4212,C 0.0619,E1 2.5487,E2 413.6085} C_DIS
LIN {X 109.4611,Y 83.1686,Z 187,A 38.2712,B 2.4211,C 0.0658,E1 2.5518,E2 415.4177} C_DIS
LIN {X 112.0557,Y 79.6381,Z 187,A 36.575,B 2.421,C 0.069,E1 2.5546,E2 417.0984} C_DIS
LIN {X 114.7979,Y 75.6306,Z 187,A 34.4804,B 2.4208,C 0.0744,E1 2.5578,E2 419.2022} C_DIS
LIN {X 120.0272,Y 67.0237,Z 187,A 30.6225,B 2.4206,C 0.082,E1 2.5633,E2 423.0195} C_DIS
LIN {X 122.2467,Y 62.8815,Z 187,A 28.8676,B 2.4205,C 0.0853,E1 2.5655,E2 424.7497} C_DIS
LIN {X 123.6606,Y 60.0564,Z 187,A 27.4548,B 2.4203,C 0.0894,E1 2.5673,E2 426.1751} C_DIS
LIN {X 126.5459,Y 53.7103,Z 187,A 24.8954,B 2.4201,C 0.0941,E1 2.5702,E2 428.6924} C_DIS
LIN {X 129.0732,Y 47.3147,Z 187,A 22.0977,B 2.4199,C 0.1011,E1 2.573,E2 431.4828} C_DIS
LIN {X 130.3449,Y 43.6842,Z 187,A 20.626,B 2.4197,C 0.1043,E1 2.5743,E2 432.9387} C_DIS
LIN {X 131.3034,Y 40.7151,Z 187,A 19.5271,B 2.4197,C 0.1062,E1 2.5752,E2 434.013} C_DIS
LIN {X 132.3621,Y 37.126,Z 187,A 17.951,B 2.4194,C 0.1105,E1 2.5764,E2 435.5918} C_DIS
LIN {X 133.1883,Y 34.0439,Z 187,A 16.6993,B 2.4194,C 0.1135,E1 2.5773,E2 436.8343} C_DIS
LIN {X 133.9706,Y 30.822,Z 187,A 15.3822,B 2.4192,C 0.1167,E1 2.5781,E2 438.1439} C_DIS
LIN {X 134.6054,Y 27.924,Z 187,A 14.313,B 2.4191,C 0.1187,E1 2.5788,E2 439.1926} C_DIS
LIN {X 135.2893,Y 24.391,Z 187,A 12.8731,B 2.4189,C 0.1224,E1 2.5795,E2 440.6257} C_DIS
LIN {X 135.8453,Y 21.0749,Z 187,A 11.4547,B 2.4187,C 0.1264,E1 2.5801,E2 442.047} C_DIS
LIN {X 136.6528,Y 14.9726,Z 187,A 8.9235,B 2.4183,C 0.1333,E1 2.581,E2 444.5753} C_DIS
LIN {X 137.0093,Y 11.2556,Z 187,A 6.9803,B 2.4179,C 0.1409,E1 2.5815,E2 446.5684} C_DIS
LIN {X 137.3364,Y 6.1173,Z 187,A 5.4222,B 2.4179,C 0.142,E1 2.5817,E2 448.0534} C_DIS
LIN {X 137.4503,Y 2.3652,Z 187,A 4.0425,B 2.4176,C 0.1448,E1 2.5817,E2 449.4104} C_DIS
LIN {X 137.4465,Y -2.5945,Z 187,A 1.6601,B 2.4171,C 0.1533,E1 2.5817,E2 451.8343} C_DIS
LIN {X 137.3007,Y -6.8311,Z 187,A 0.3406,B 2.4171,C 0.1545,E1 2.5815,E2 453.0978} C_DIS
LIN {X 137.0229,Y -11.0945,Z 187,A -1.1779,B 2.4169,C 0.1572,E1 2.5812,E2 454.5839} C_DIS
LIN {X 136.7237,Y -14.3149,Z 187,A -2.4365,B 2.4167,C 0.1602,E1 2.5809,E2 455.8318} C_DIS
LIN {X 135.9635,Y -20.3116,Z 187,A -5.0222,B 2.4162,C 0.1678,E1 2.58,E2 458.4278} C_DIS
LIN {X 135.3319,Y -24.1532,Z 187,A -6.3564,B 2.416,C 0.1699,E1 2.5793,E2 459.7258} C_DIS
LIN {X 134.4144,Y -28.825,Z 187,A -8.3822,B 2.4156,C 0.1757,E1 2.5782,E2 461.7584} C_DIS
LIN {X 133.4301,Y -33.0913,Z 187,A -10.0018,B 2.4154,C 0.179,E1 2.5772,E2 463.3528} C_DIS
LIN {X 132.4659,Y -36.7547,Z 187,A -11.5496,B 2.415,C 0.183,E1 2.5761,E2 464.8976} C_DIS
LIN {X 131.5659,Y -39.8575,Z 187,A -12.8023,B 2.4148,C 0.1859,E1 2.5751,E2 466.1391} C_DIS
LIN {X 130.7644,Y -42.4156,Z 187,A -13.9054,B 2.4146,C 0.1888,E1 2.5741,E2 467.2413} C_DIS
LIN {X 129.7401,Y -45.4502,Z 187,A -15.0834,B 2.4144,C 0.191,E1 2.5731,E2 468.3997} C_DIS
LIN {X 128.4443,Y -48.9976,Z 187,A -16.7423,B 2.414,C 0.1959,E1 2.5714,E2 470.071} C_DIS
LIN {X 126.9667,Y -52.7026,Z 187,A -18.0895,B 2.4139,C 0.1977,E1 2.5701,E2 471.3781} C_DIS
LIN {X 125.6228,Y -55.8304,Z 187,A -19.5515,B 2.4136,C 0.2017,E1 2.5684,E2 472.8469} C_DIS
LIN {X 124.1504,Y -59.0318,Z 187,A -20.9376,B 2.4133,C 0.2048,E1 2.5668,E2 474.2233} C_DIS
LIN {X 122.7146,Y -61.9623,Z 187,A -22.1198,B 2.4131,C 0.2068,E1 2.5654,E2 475.3832} C_DIS
LIN {X 120.9266,Y -65.387,Z 187,A -24.1498,B 2.4125,C 0.2144,E1 2.5626,E2 477.4695} C_DIS
LIN {X 119.0017,Y -68.827,Z 187,A -25.3497,B 2.4125,C 0.2148,E1 2.561,E2 478.6126} C_DIS
LIN {X 116.9068,Y -72.3291,Z 187,A -27.0454,B 2.4121,C 0.2189,E1 2.5586,E2 480.309} C_DIS
LIN {X 114.8014,Y -75.6253,Z 187,A -28.8389,B 2.4116,C 0.2242,E1 2.5558,E2 482.1252} C_DIS
LIN {X 112.6999,Y -78.7232,Z 187,A -30.0217,B 2.4116,C 0.2248,E1 2.554,E2 483.2596} C_DIS
LIN {X 110.2655,Y -82.0979,Z 187,A -31.7054,B 2.4112,C 0.2285,E1 2.5512,E2 484.938} C_DIS
LIN {X 107.5124,Y -85.6717,Z 187,A -33.463,B 2.4109,C 0.2318,E1 2.5482,E2 486.6808} C_DIS
LIN {X 104.4569,Y -89.3728,Z 187,A -35.2688,B 2.4106,C 0.2347,E1 2.545,E2 488.4624} C_DIS
LIN {X 100.872,Y -93.3999,Z 187,A -37.5199,B 2.4101,C 0.2396,E1 2.5408,E2 490.7158} C_DIS
LIN {X 98.075,Y -96.332,Z 187,A -39.3254,B 2.4096,C 0.2441,E1 2.5373,E2 492.5381} C_DIS
LIN {X 94.3006,Y -100.0298,Z 187,A -41.2942,B 2.4094,C 0.2468,E1 2.5334,E2 494.4776} C_DIS
LIN {X 90.5568,Y -103.4315,Z 187,A -43.3345,B 2.409,C 0.2504,E1 2.5291,E2 496.5105} C_DIS
LIN {X 87.1737,Y -106.2984,Z 187,A -45.1616,B 2.4086,C 0.2538,E1 2.5252,E2 498.3362} C_DIS
LIN {X 83.6074,Y -109.1255,Z 187,A -46.8897,B 2.4084,C 0.256,E1 2.5214,E2 500.0432} C_DIS
LIN {X 79.5573,Y -112.1131,Z 187,A -48.9822,B 2.408,C 0.2597,E1 2.5167,E2 502.1367} C_DIS
LIN {X 76.1596,Y -114.4479,Z 187,A -50.5916,B 2.4078,C 0.2618,E1 2.513,E2 503.7328} C_DIS
LIN {X 72.9438,Y -116.5242,Z 187,A -52.094,B 2.4076,C 0.2637,E1 2.5095,E2 505.224} C_DIS
LIN {X 66.769,Y -120.1687,Z 187,A -55.0115,B 2.4071,C 0.2679,E1 2.5025,E2 508.1342} C_DIS
LIN {X 63.6382,Y -121.8534,Z 187,A -56.2969,B 2.4071,C 0.2686,E1 2.4993,E2 509.3942} C_DIS
LIN {X 61.4031,Y -122.9963,Z 187,A -57.3507,B 2.4069,C 0.2702,E1 2.4967,E2 510.4498} C_DIS
LIN {X 58.5788,Y -124.3668,Z 187,A -58.7376,B 2.4066,C 0.2725,E1 2.4932,E2 511.8482} C_DIS
LIN {X 55.0185,Y -125.9811,Z 187,A -60.2911,B 2.4064,C 0.2741,E1 2.4892,E2 513.3926} C_DIS
LIN {X 51.726,Y -127.3678,Z 187,A -61.5414,B 2.4064,C 0.2743,E1 2.4861,E2 514.6118} C_DIS
LIN {X 49.2715,Y -128.3381,Z 187,A -62.9906,B 2.406,C 0.278,E1 2.4822,E2 516.1088} C_DIS
LIN {X 44.2109,Y -130.1695,Z 187,A -65.0848,B 2.4058,C 0.2795,E1 2.4767,E2 518.1845} C_DIS
LIN {X 40.7652,Y -131.2881,Z 187,A -66.3565,B 2.4058,C 0.2795,E1 2.4734,E2 519.425} C_DIS
LIN {X 37.2172,Y -132.3366,Z 187,A -67.9696,B 2.4056,C 0.2814,E1 2.469,E2 521.0487} C_DIS
LIN {X 34.4029,Y -133.0972,Z 187,A -69.2115,B 2.4054,C 0.2827,E1 2.4657,E2 522.295} C_DIS
LIN {X 30.766,Y -133.9834,Z 187,A -70.6815,B 2.4054,C 0.2834,E1 2.4617,E2 523.7538} C_DIS
LIN {X 27.8265,Y -134.6252,Z 187,A -71.8111,B 2.4054,C 0.2835,E1 2.4586,E2 524.8673} C_DIS
LIN {X 24.297,Y -135.3062,Z 187,A -74.6781,B 2.4042,C 0.2933,E1 2.4503,E2 527.9185} C_DIS
LIN {X 15.6267,Y -136.581,Z 187,A -77.88,B 2.4042,C 0.2924,E1 2.4415,E2 531.0626} C_DIS
LIN {X 9.1847,Y -137.1653,Z 187,A -79.973,B 2.4046,C 0.2899,E1 2.4359,E2 533.0763} C_DIS
LIN {X 5.9846,Y -137.3415,Z 187,A -81.4073,B 2.4044,C 0.2909,E1 2.4318,E2 534.5245} C_DIS
LIN {X 2.2221,Y -137.4527,Z 187,A -82.6131,B 2.4047,C 0.2891,E1 2.4286,E2 535.6821} C_DIS
LIN {X 2.2221,Y -137.4527,Z 187,A -82.6131,B 2.4047,C 0.2891,E1 2.4286,E2 535.6821} C_DIS
Enddeposition()
LIN {X 0.9823,Y -138.3652,Z 187,A -82.5702,B 2.4082,C 0.2873,E1 2.4321,E2 535.5922} C_DIS
Startdeposition()
$VEL.CP = VEL_PRINT
LIN {X 4.6169,Y -138.2954,Z 187,A -80.9818,B 2.4082,C 0.2864,E1 2.4366,E2 533.9918} C_DIS
LIN {X 7.7265,Y -138.1565,Z 187,A -79.6907,B 2.4083,C 0.286,E1 2.4402,E2 532.6996} C_DIS
LIN {X 10.8859,Y -137.9434,Z 187,A -78.3969,B 2.4083,C 0.2855,E1 2.4438,E2 531.4076} C_DIS
LIN {X 14.5972,Y -137.5982,Z 187,A -76.8938,B 2.4084,C 0.2851,E1 2.448,E2 529.9092} C_DIS
LIN {X 17.2115,Y -137.2977,Z 187,A -75.7869,B 2.4085,C 0.2844,E1 2.451,E2 528.7993} C_DIS
LIN {X 20.3995,Y -136.8603,Z 187,A -74.4684,B 2.4085,C 0.2837,E1 2.4547,E2 527.4819} C_DIS
LIN {X 23.601,Y -136.3447,Z 187,A -73.1516,B 2.4087,C 0.2829,E1 2.4583,E2 526.168} C_DIS
LIN {X 26.786,Y -135.7551,Z 187,A -71.8082,B 2.4087,C 0.282,E1 2.462,E2 524.8235} C_DIS
LIN {X 30.4491,Y -134.9786,Z 187,A -70.2529,B 2.4089,C 0.2807,E1 2.4663,E2 523.2665} C_DIS
LIN {X 33.2322,Y -134.3226,Z 187,A -69.1253,B 2.409,C 0.2801,E1 2.4693,E2 522.1459} C_DIS
LIN {X 36.4878,Y -133.4748,Z 187,A -67.7564,B 2.4091,C 0.279,E1 2.473,E2 520.7794} C_DIS
LIN {X 39.7152,Y -132.5503,Z 187,A -66.2605,B 2.4094,C 0.2769,E1 2.4771,E2 519.2682} C_DIS
LIN {X 42.9845,Y -131.5262,Z 187,A -65.029,B 2.4094,C 0.2767,E1 2.4803,E2 518.0614} C_DIS
LIN {X 46.1286,Y -130.4572,Z 187,A -63.6559,B 2.4096,C 0.2752,E1 2.4839,E2 516.6877} C_DIS
LIN {X 49.6949,Y -129.1388,Z 187,A -62.1178,B 2.4097,C 0.2736,E1 2.4879,E2 515.1534} C_DIS
LIN {X 52.5291,Y -128.0141,Z 187,A -60.7467,B 2.41,C 0.2713,E1 2.4915,E2 513.7667} C_DIS
LIN {X 55.733,Y -126.6519,Z 187,A -59.4785,B 2.41,C 0.2707,E1 2.4947,E2 512.5213} C_DIS
LIN {X 58.863,Y -125.2281,Z 187,A -58.0923,B 2.4103,C 0.2691,E1 2.4982,E2 511.1392} C_DIS
LIN {X 62.0232,Y -123.6932,Z 187,A -56.6773,B 2.4105,C 0.2673,E1 2.5018,E2 509.7286} C_DIS
LIN {X 65.6782,Y -121.7914,Z 187,A -54.994,B 2.4107,C 0.265,E1 2.5059,E2 508.0471} C_DIS
LIN {X 68.9575,Y -119.9657,Z 187,A -53.5133,B 2.4109,C 0.2632,E1 2.5095,E2 506.5754} C_DIS
LIN {X 71.979,Y -118.1776,Z 187,A -52.1052,B 2.4111,C 0.2612,E1 2.5129,E2 505.1725} C_DIS
LIN {X 74.9885,Y -116.2912,Z 187,A -50.6823,B 2.4113,C 0.2591,E1 2.5162,E2 503.755} C_DIS
LIN {X 77.9316,Y -114.3398,Z 187,A -49.1594,B 2.4117,C 0.2562,E1 2.5198,E2 502.2226} C_DIS
LIN {X 81.576,Y -111.7688,Z 187,A -47.4911,B 2.4119,C 0.2543,E1 2.5235,E2 500.5773} C_DIS
LIN {X 84.4155,Y -109.6401,Z 187,A -46.067,B 2.4121,C 0.252,E1 2.5267,E2 499.1583} C_DIS
LIN {X 87.2276,Y -107.4162,Z 187,A -44.6418,B 2.4123,C 0.2496,E1 2.5298,E2 497.74} C_DIS
LIN {X 90.3645,Y -104.7902,Z 187,A -42.9613,B 2.4127,C 0.2465,E1 2.5333,E2 496.06} C_DIS
LIN {X 93.3132,Y -102.1742,Z 187,A -41.4452,B 2.4129,C 0.2441,E1 2.5365,E2 494.5585} C_DIS
LIN {X 95.937,Y -99.7146,Z 187,A -40.0165,B 2.4132,C 0.2416,E1 2.5393,E2 493.1368} C_DIS
LIN {X 98.4753,Y -97.2088,Z 187,A -38.5971,B 2.4134,C 0.239,E1 2.5421,E2 491.724} C_DIS
LIN {X 101.2504,Y -94.3137,Z 187,A -36.9456,B 2.4138,C 0.2355,E1 2.5453,E2 490.0724} C_DIS
LIN {X 104.0313,Y -91.2378,Z 187,A -35.3947,B 2.414,C 0.2331,E1 2.5481,E2 488.5427} C_DIS
LIN {X 106.2907,Y -88.5958,Z 187,A -33.9936,B 2.4143,C 0.2302,E1 2.5507,E2 487.1456} C_DIS
LIN {X 108.5424,Y -85.8223,Z 187,A -32.4723,B 2.4146,C 0.2265,E1 2.5533,E2 485.6175} C_DIS
LIN {X 111.2506,Y -82.2814,Z 187,A -30.821,B 2.4149,C 0.2238,E1 2.5561,E2 483.991} C_DIS
LIN {X 113.4849,Y -79.1702,Z 187,A -29.3771,B 2.4151,C 0.2213,E1 2.5584,E2 482.5649} C_DIS
LIN {X 115.5021,Y -76.1972,Z 187,A -27.8082,B 2.4155,C 0.217,E1 2.5608,E2 480.984} C_DIS
LIN {X 117.9911,Y -72.283,Z 187,A -26.0206,B 2.4158,C 0.2135,E1 2.5634,E2 479.2127} C_DIS
LIN {X 119.9732,Y -68.9446,Z 187,A -24.426,B 2.4162,C 0.2096,E1 2.5657,E2 477.6187} C_DIS
Enddeposition()
END
